C03642=1224.310,-102.269,-36.664,179.469,5.331,149.087
C03643=1224.305,-102.020,-36.674,179.472,5.331,149.087
C03644=1224.300,-101.770,-36.685,179.474,5.331,149.086
C03645=1224.294,-101.520,-36.695,179.476,5.332,149.085
C03646=1224.289,-101.271,-36.706,179.478,5.331,149.085
C03647=1224.283,-100.999,-36.717,179.481,5.332,149.084
C03648=1224.278,-100.728,-36.728,179.484,5.331,149.083
C03649=1224.272,-100.457,-36.740,179.486,5.331,149.082
C03650=1224.266,-100.186,-36.751,179.489,5.332,149.082
C03651=1224.261,-99.936,-36.761,179.491,5.331,149.081
C03652=1224.256,-99.687,-36.772,179.494,5.332,149.080
C03653=1224.251,-99.437,-36.783,179.496,5.332,149.079
C03654=1224.245,-99.187,-36.793,179.498,5.332,149.079
C03655=1224.240,-98.937,-36.804,179.500,5.332,149.078
C03656=1224.235,-98.688,-36.814,179.503,5.332,149.078
C03657=1224.230,-98.438,-36.825,179.505,5.332,149.077
C03658=1224.225,-98.189,-36.835,179.507,5.332,149.076
C03659=1224.220,-97.938,-36.846,179.510,5.332,149.075
C03660=1224.214,-97.689,-36.857,179.512,5.332,149.075
C03661=1224.209,-97.439,-36.868,179.514,5.332,149.074
C03662=1224.204,-97.190,-36.878,179.516,5.332,149.073
C03663=1224.199,-96.939,-36.888,179.519,5.332,149.073
C03664=1224.193,-96.690,-36.899,179.521,5.332,149.072
C03665=1224.188,-96.440,-36.910,179.523,5.333,149.071
C03666=1224.183,-96.191,-36.920,179.525,5.332,149.071
C03667=1224.178,-95.941,-36.931,179.528,5.333,149.070
C03668=1224.173,-95.691,-36.942,179.530,5.332,149.069
C03669=1224.168,-95.441,-36.952,179.533,5.333,149.069
C03670=1224.162,-95.192,-36.963,179.535,5.332,149.068
C03671=1224.157,-94.942,-36.974,179.538,5.333,149.067
C03672=1224.152,-94.692,-36.984,179.540,5.333,149.066
C03673=1224.147,-94.443,-36.995,179.542,5.333,149.066
C03674=1224.141,-94.193,-37.006,179.544,5.333,149.065
C03675=1224.136,-93.943,-37.016,179.547,5.333,149.064
C03676=1224.130,-93.694,-37.027,179.549,5.333,149.064
C03677=1224.125,-93.444,-37.038,179.551,5.334,149.063
C03678=1224.120,-93.195,-37.049,179.554,5.333,149.062
C03679=1224.115,-92.944,-37.059,179.556,5.334,149.062
C03680=1224.110,-92.694,-37.070,179.558,5.333,149.061
C03681=1224.105,-92.445,-37.081,179.561,5.334,149.060
C03682=1224.100,-92.195,-37.092,179.563,5.333,149.059
C03683=1224.094,-91.946,-37.102,179.566,5.334,149.059
C03684=1224.089,-91.696,-37.114,179.568,5.333,149.058
C03685=1224.083,-91.446,-37.124,179.571,5.334,149.057
C03686=1224.078,-91.196,-37.135,179.573,5.334,149.057
C03687=1224.073,-90.946,-37.146,179.575,5.334,149.056
C03688=1224.068,-90.697,-37.157,179.577,5.334,149.055
C03689=1224.063,-90.447,-37.167,179.580,5.334,149.055
C03690=1224.058,-90.198,-37.178,179.582,5.334,149.054
C03691=1224.053,-89.948,-37.189,179.584,5.334,149.053
C03692=1224.047,-89.698,-37.201,179.586,5.334,149.053
C03693=1224.042,-89.448,-37.211,179.589,5.335,149.052
C03694=1224.037,-89.199,-37.222,179.591,5.334,149.051
C03695=1224.032,-88.949,-37.232,179.594,5.335,149.050
C03696=1224.027,-88.699,-37.244,179.596,5.334,149.050
C03697=1224.022,-88.449,-37.254,179.599,5.335,149.049
C03698=1224.016,-88.200,-37.266,179.601,5.334,149.048
C03699=1224.011,-87.950,-37.276,179.603,5.335,149.048
C03700=1224.006,-87.701,-37.287,179.605,5.334,149.047
C03701=1224.001,-87.451,-37.298,179.608,5.335,149.046
C03702=1223.996,-87.201,-37.309,179.610,5.335,149.046
C03703=1223.990,-86.952,-37.321,179.612,5.335,149.045
C03704=1223.985,-86.701,-37.331,179.614,5.335,149.044
C03705=1223.980,-86.452,-37.342,179.617,5.335,149.044
C03706=1223.975,-86.202,-37.353,179.619,5.335,149.043
C03707=1223.969,-85.952,-37.365,179.622,5.336,149.042
C03708=1223.964,-85.703,-37.376,179.624,5.335,149.041
C03709=1223.959,-85.453,-37.386,179.627,5.336,149.041
C03710=1223.954,-85.204,-37.397,179.629,5.335,149.040
C03711=1223.949,-84.953,-37.408,179.631,5.336,149.039
C03712=1223.943,-84.704,-37.419,179.634,5.335,149.039
C03713=1223.938,-84.454,-37.431,179.636,5.336,149.038
C03714=1223.933,-84.204,-37.441,179.638,5.335,149.037
C03715=1223.927,-83.955,-37.453,179.641,5.336,149.036
C03716=1223.923,-83.705,-37.464,179.644,5.336,149.036
C03717=1223.918,-83.455,-37.475,179.645,5.336,149.035
C03718=1223.912,-83.206,-37.486,179.648,5.337,149.035
C03719=1223.907,-82.956,-37.497,179.650,5.337,149.034
C03720=1223.902,-82.706,-37.508,179.653,5.337,149.033
C03721=1223.897,-82.457,-37.519,179.655,5.337,149.032
C03722=1223.892,-82.207,-37.530,179.657,5.337,149.032
C03723=1223.886,-81.957,-37.541,179.660,5.337,149.031
C03724=1223.882,-81.707,-37.553,179.662,5.337,149.030
C03725=1223.876,-81.458,-37.564,179.664,5.337,149.030
C03726=1223.870,-81.208,-37.575,179.667,5.337,149.029
C03727=1223.866,-80.958,-37.586,179.669,5.337,149.028
C03728=1223.861,-80.709,-37.597,179.672,5.337,149.027
C03729=1223.855,-80.459,-37.609,179.674,5.337,149.027
C03730=1223.850,-80.209,-37.620,179.676,5.337,149.026
C03731=1223.845,-79.959,-37.631,179.679,5.337,149.025
C03732=1223.839,-79.710,-37.642,179.681,5.338,149.025
C03733=1223.835,-79.461,-37.654,179.683,5.337,149.024
C03734=1223.829,-79.211,-37.665,179.686,5.338,149.023
C03735=1223.824,-78.961,-37.676,179.688,5.338,149.023
C03736=1223.819,-78.711,-37.687,179.690,5.338,149.022
C03737=1223.814,-78.462,-37.699,179.692,5.338,149.021
C03738=1223.809,-78.212,-37.710,179.695,5.338,149.021
C03739=1223.804,-77.963,-37.721,179.697,5.338,149.020
C03740=1223.798,-77.712,-37.732,179.700,5.338,149.019
C03741=1223.793,-77.463,-37.744,179.702,5.339,149.018
C03742=1223.788,-77.213,-37.755,179.705,5.338,149.018
C03743=1223.783,-76.963,-37.767,179.707,5.339,149.017
C03744=1223.778,-76.714,-37.778,179.709,5.339,149.016
C03745=1223.772,-76.464,-37.790,179.712,5.339,149.016
C03746=1223.767,-76.214,-37.800,179.714,5.339,149.015
C03747=1223.762,-75.964,-37.812,179.717,5.339,149.014
C03748=1223.757,-75.715,-37.823,179.719,5.339,149.014
C03749=1223.751,-75.465,-37.835,179.722,5.339,149.013
C03750=1223.746,-75.216,-37.846,179.724,5.339,149.012
C03751=1223.741,-74.945,-37.858,179.726,5.339,149.011
C03752=1223.735,-74.675,-37.871,179.729,5.340,149.011
C03753=1223.729,-74.404,-37.883,179.731,5.339,149.010
C03754=1223.723,-74.134,-37.896,179.734,5.339,149.009
C03755=1223.719,-73.885,-37.907,179.736,5.339,149.009
C03756=1223.713,-73.635,-37.919,179.738,5.340,149.008
C03757=1223.708,-73.385,-37.930,179.741,5.340,149.007
C03758=1223.703,-73.135,-37.941,179.743,5.340,149.006
C03759=1223.698,-72.885,-37.953,179.746,5.341,149.006
C03760=1223.692,-72.636,-37.964,179.748,5.340,149.005
C03761=1223.687,-72.386,-37.976,179.751,5.341,149.004
C03762=1223.682,-72.136,-37.987,179.753,5.340,149.004
C03763=1223.677,-71.887,-37.999,179.755,5.341,149.003
C03764=1223.672,-71.637,-38.011,179.758,5.340,149.002
C03765=1223.667,-71.387,-38.022,179.760,5.341,149.001
C03766=1223.661,-71.138,-38.033,179.762,5.340,149.001
C03767=1223.656,-70.888,-38.045,179.765,5.341,149.000
C03768=1223.651,-70.638,-38.057,179.768,5.341,148.999
C03769=1223.646,-70.389,-38.068,179.770,5.341,148.999
C03770=1223.641,-70.139,-38.080,179.772,5.342,148.998
C03771=1223.635,-69.889,-38.092,179.774,5.341,148.997
C03772=1223.630,-69.640,-38.103,179.777,5.342,148.997
C03773=1223.625,-69.390,-38.114,179.779,5.341,148.996
C03774=1223.620,-69.141,-38.126,179.782,5.342,148.995
C03775=1223.615,-68.891,-38.138,179.784,5.341,148.994
C03776=1223.610,-68.641,-38.150,179.787,5.342,148.994
C03777=1223.605,-68.391,-38.162,179.789,5.342,148.993
C03778=1223.599,-68.142,-38.173,179.791,5.342,148.992
C03779=1223.595,-67.892,-38.185,179.794,5.342,148.992
C03780=1223.589,-67.642,-38.197,179.796,5.342,148.991
C03781=1223.584,-67.393,-38.207,179.799,5.343,148.990
C03782=1223.579,-67.143,-38.219,179.800,5.343,148.990
C03783=1223.573,-66.893,-38.231,179.803,5.343,148.989
C03784=1223.569,-66.644,-38.243,179.805,5.343,148.988
C03785=1223.563,-66.394,-38.255,179.808,5.343,148.988
C03786=1223.559,-66.145,-38.266,179.810,5.343,148.987
C03787=1223.553,-65.895,-38.278,179.813,5.343,148.986
C03788=1223.548,-65.645,-38.290,179.815,5.343,148.985
C03789=1223.543,-65.395,-38.302,179.817,5.343,148.985
C03790=1223.538,-65.145,-38.313,179.820,5.344,148.984
C03791=1223.532,-64.896,-38.326,179.822,5.344,148.983
C03792=1223.527,-64.647,-38.337,179.825,5.344,148.983
C03793=1223.522,-64.397,-38.349,179.827,5.344,148.982
C03794=1223.516,-64.147,-38.361,179.830,5.344,148.981
C03795=1223.512,-63.897,-38.372,179.832,5.344,148.981
C03796=1223.507,-63.648,-38.385,179.834,5.344,148.980
C03797=1223.501,-63.398,-38.396,179.837,5.345,148.979
C03798=1223.496,-63.149,-38.408,179.839,5.344,148.978
C03799=1223.491,-62.899,-38.420,179.842,5.345,148.978
C03800=1223.486,-62.649,-38.432,179.844,5.344,148.977
C03801=1223.480,-62.399,-38.444,179.846,5.345,148.976
C03802=1223.476,-62.150,-38.455,179.849,5.345,148.976
C03803=1223.470,-61.900,-38.467,179.851,5.345,148.975
C03804=1223.465,-61.650,-38.480,179.853,5.345,148.974
C03805=1223.460,-61.401,-38.491,179.856,5.345,148.973
C03806=1223.455,-61.151,-38.503,179.859,5.346,148.973
C03807=1223.450,-60.902,-38.516,179.861,5.345,148.972
C03808=1223.445,-60.652,-38.528,179.863,5.346,148.971
C03809=1223.440,-60.402,-38.539,179.865,5.345,148.971
C03810=1223.434,-60.152,-38.551,179.868,5.346,148.970
C03811=1223.429,-59.903,-38.563,179.870,5.346,148.969
C03812=1223.424,-59.653,-38.575,179.873,5.346,148.969
C03813=1223.419,-59.403,-38.587,179.876,5.347,148.968
C03814=1223.414,-59.154,-38.599,179.878,5.346,148.967
C03815=1223.409,-58.904,-38.611,179.880,5.347,148.966
C03816=1223.403,-58.655,-38.624,179.882,5.346,148.966
C03817=1223.399,-58.405,-38.635,179.885,5.347,148.965
C03818=1223.393,-58.155,-38.647,179.887,5.346,148.964
C03819=1223.388,-57.906,-38.659,179.890,5.347,148.964
C03820=1223.383,-57.656,-38.671,179.893,5.347,148.963
C03821=1223.377,-57.406,-38.683,179.895,5.347,148.962
C03822=1223.373,-57.157,-38.695,179.897,5.348,148.962
C03823=1223.368,-56.907,-38.707,179.899,5.348,148.961
C03824=1223.362,-56.658,-38.720,179.902,5.348,148.960
C03825=1223.357,-56.408,-38.732,179.904,5.348,148.960
C03826=1223.352,-56.158,-38.744,179.906,5.348,148.959
C03827=1223.346,-55.908,-38.756,179.909,5.349,148.958
C03828=1223.342,-55.659,-38.767,179.911,5.348,148.957
C03829=1223.337,-55.409,-38.780,179.914,5.349,148.957
C03830=1223.332,-55.159,-38.792,179.916,5.348,148.956
C03831=1223.327,-54.910,-38.805,179.918,5.349,148.955
C03832=1223.321,-54.660,-38.817,179.921,5.349,148.955
C03833=1223.316,-54.410,-38.829,179.923,5.349,148.954
C03834=1223.311,-54.161,-38.841,179.926,5.350,148.953
C03835=1223.306,-53.911,-38.853,179.928,5.349,148.953
C03836=1223.301,-53.661,-38.865,179.931,5.350,148.952
C03837=1223.296,-53.412,-38.878,179.933,5.349,148.951
C03838=1223.290,-53.162,-38.889,179.935,5.350,148.950
C03839=1223.285,-52.913,-38.902,179.938,5.350,148.950
C03840=1223.280,-52.662,-38.914,179.940,5.350,148.949
C03841=1223.275,-52.413,-38.927,179.943,5.350,148.948
C03842=1223.270,-52.163,-38.939,179.945,5.350,148.948
C03843=1223.265,-51.914,-38.951,179.948,5.351,148.947
C03844=1223.260,-51.665,-38.963,179.950,5.351,148.946
C03845=1223.255,-51.415,-38.975,179.952,5.351,148.946
C03846=1223.250,-51.165,-38.988,179.955,5.351,148.945
C03847=1223.244,-50.915,-39.000,179.957,5.351,148.944
C03848=1223.239,-50.666,-39.012,179.960,5.351,148.943
C03849=1223.234,-50.415,-39.025,179.962,5.352,148.943
C03850=1223.229,-50.166,-39.037,179.964,5.351,148.942
C03851=1223.224,-49.917,-39.050,179.967,5.352,148.941
C03852=1223.219,-49.667,-39.062,179.969,5.352,148.941
C03853=1223.214,-49.418,-39.074,179.972,5.352,148.940
C03854=1223.208,-49.168,-39.087,179.975,5.353,148.939
C03855=1223.203,-48.898,-39.100,179.977,5.352,148.938
C03856=1223.197,-48.628,-39.114,179.979,5.353,148.938
C03857=1223.191,-48.358,-39.127,179.982,5.353,148.937
C03858=1223.186,-48.088,-39.140,179.985,5.352,148.936
C03859=1223.181,-47.839,-39.153,179.987,5.353,148.935
C03860=1223.176,-47.589,-39.165,179.990,5.353,148.935
C03861=1223.171,-47.340,-39.178,179.992,5.353,148.934
C03862=1223.166,-47.090,-39.191,179.995,5.354,148.933
C03863=1223.161,-46.840,-39.202,179.997,5.353,148.933
C03864=1223.156,-46.591,-39.215,179.999,5.354,148.932
C03865=1223.151,-46.341,-39.228,-179.998,5.354,148.931
C03866=1223.145,-46.091,-39.239,-179.996,5.354,148.931
C03867=1223.140,-45.842,-39.252,-179.993,5.354,148.930
C03868=1223.136,-45.592,-39.265,-179.991,5.354,148.929
C03869=1223.130,-45.343,-39.278,-179.988,5.354,148.928
C03870=1223.124,-45.092,-39.290,-179.986,5.355,148.928
C03871=1223.119,-44.843,-39.303,-179.984,5.355,148.927
C03872=1223.114,-44.594,-39.315,-179.981,5.355,148.926
C03873=1223.109,-44.344,-39.328,-179.978,5.356,148.926
C03874=1223.104,-44.094,-39.340,-179.976,5.355,148.925
C03875=1223.099,-43.845,-39.353,-179.974,5.356,148.924
C03876=1223.094,-43.595,-39.365,-179.972,5.355,148.924
C03877=1223.089,-43.345,-39.378,-179.969,5.356,148.923
C03878=1223.084,-43.096,-39.391,-179.966,5.356,148.922
C03879=1223.079,-42.846,-39.403,-179.964,5.356,148.921
C03880=1223.074,-42.597,-39.415,-179.961,5.357,148.921
C03881=1223.068,-42.346,-39.429,-179.959,5.356,148.920
C03882=1223.063,-42.097,-39.442,-179.957,5.357,148.919
C03883=1223.058,-41.848,-39.454,-179.954,5.357,148.919
C03884=1223.053,-41.598,-39.467,-179.952,5.357,148.918
C03885=1223.048,-41.348,-39.480,-179.949,5.357,148.917
C03886=1223.043,-41.098,-39.492,-179.947,5.358,148.916
C03887=1223.038,-40.849,-39.504,-179.945,5.358,148.916
C03888=1223.032,-40.599,-39.517,-179.942,5.358,148.915
C03889=1223.027,-40.349,-39.530,-179.940,5.358,148.914
C03890=1223.022,-40.100,-39.543,-179.937,5.358,148.914
C03891=1223.017,-39.851,-39.556,-179.934,5.359,148.913
C03892=1223.012,-39.602,-39.568,-179.932,5.358,148.912
C03893=1223.008,-39.351,-39.581,-179.930,5.359,148.912
C03894=1223.002,-39.102,-39.594,-179.927,5.359,148.911
C03895=1222.997,-38.853,-39.607,-179.925,5.359,148.910
C03896=1222.992,-38.602,-39.619,-179.923,5.360,148.910
C03897=1222.987,-38.353,-39.632,-179.921,5.359,148.909
C03898=1222.982,-38.103,-39.644,-179.918,5.360,148.908
C03899=1222.976,-37.854,-39.658,-179.915,5.360,148.908
C03900=1222.971,-37.604,-39.671,-179.913,5.360,148.907
C03901=1222.966,-37.354,-39.683,-179.911,5.361,148.906
C03902=1222.961,-37.105,-39.696,-179.908,5.361,148.906
C03903=1222.956,-36.855,-39.709,-179.906,5.361,148.905
C03904=1222.951,-36.605,-39.722,-179.903,5.361,148.904
C03905=1222.945,-36.356,-39.735,-179.901,5.361,148.903
C03906=1222.941,-36.106,-39.748,-179.899,5.361,148.903
C03907=1222.935,-35.856,-39.761,-179.896,5.362,148.902
C03908=1222.930,-35.607,-39.773,-179.894,5.362,148.901
C03909=1222.925,-35.357,-39.786,-179.891,5.362,148.901
C03910=1222.920,-35.108,-39.799,-179.888,5.363,148.900
C03911=1222.914,-34.858,-39.812,-179.886,5.362,148.899
C03912=1222.910,-34.609,-39.826,-179.884,5.363,148.899
C03913=1222.905,-34.359,-39.838,-179.881,5.363,148.898
C03914=1222.899,-34.110,-39.852,-179.879,5.363,148.897
C03915=1222.895,-33.860,-39.865,-179.876,5.363,148.896
C03916=1222.890,-33.610,-39.877,-179.874,5.364,148.896
C03917=1222.884,-33.361,-39.890,-179.872,5.364,148.895
C03918=1222.879,-33.111,-39.903,-179.869,5.364,148.894
C03919=1222.874,-32.861,-39.916,-179.867,5.364,148.894
C03920=1222.870,-32.611,-39.929,-179.864,5.364,148.893
C03921=1222.864,-32.362,-39.942,-179.861,5.365,148.892
C03922=1222.859,-32.113,-39.955,-179.859,5.364,148.892
C03923=1222.854,-31.863,-39.968,-179.857,5.365,148.891
C03924=1222.848,-31.613,-39.982,-179.854,5.365,148.890
C03925=1222.843,-31.364,-39.994,-179.852,5.365,148.889
C03926=1222.838,-31.114,-40.008,-179.849,5.366,148.889
C03927=1222.833,-30.864,-40.020,-179.847,5.366,148.888
C03928=1222.829,-30.615,-40.034,-179.845,5.366,148.887
C03929=1222.823,-30.365,-40.047,-179.842,5.366,148.887
C03930=1222.818,-30.116,-40.060,-179.839,5.367,148.886
C03931=1222.813,-29.866,-40.073,-179.837,5.366,148.885
C03932=1222.807,-29.617,-40.086,-179.835,5.367,148.885
C03933=1222.803,-29.367,-40.100,-179.832,5.367,148.884
C03934=1222.797,-29.117,-40.113,-179.830,5.367,148.883
C03935=1222.793,-28.867,-40.126,-179.827,5.368,148.882
C03936=1222.788,-28.618,-40.138,-179.824,5.368,148.882
C03937=1222.782,-28.369,-40.152,-179.822,5.368,148.881
C03938=1222.778,-28.119,-40.165,-179.820,5.368,148.880
C03939=1222.772,-27.869,-40.178,-179.817,5.369,148.880
C03940=1222.767,-27.619,-40.191,-179.815,5.368,148.879
C03941=1222.762,-27.370,-40.205,-179.812,5.369,148.878
C03942=1222.757,-27.120,-40.218,-179.810,5.369,148.878
C03943=1222.752,-26.871,-40.231,-179.808,5.369,148.877
C03944=1222.747,-26.621,-40.244,-179.805,5.370,148.876
C03945=1222.742,-26.372,-40.258,-179.802,5.370,148.875
C03946=1222.737,-26.122,-40.271,-179.800,5.370,148.875
C03947=1222.731,-25.872,-40.284,-179.798,5.370,148.874
C03948=1222.727,-25.623,-40.298,-179.795,5.371,148.873
C03949=1222.721,-25.373,-40.311,-179.793,5.370,148.873
C03950=1222.716,-25.124,-40.324,-179.790,5.371,148.872
C03951=1222.711,-24.874,-40.338,-179.787,5.371,148.871
C03952=1222.705,-24.625,-40.351,-179.785,5.371,148.871
C03953=1222.701,-24.375,-40.364,-179.783,5.372,148.870
C03954=1222.695,-24.126,-40.378,-179.780,5.372,148.869
C03955=1222.691,-23.876,-40.391,-179.778,5.372,148.869
C03956=1222.685,-23.627,-40.405,-179.775,5.372,148.868
C03957=1222.681,-23.377,-40.418,-179.773,5.373,148.867
C03958=1222.675,-23.127,-40.431,-179.771,5.372,148.866
C03959=1222.670,-22.858,-40.445,-179.768,5.373,148.866
C03960=1222.665,-22.589,-40.460,-179.765,5.373,148.865
C03961=1222.659,-22.318,-40.474,-179.762,5.374,148.864
C03962=1222.653,-22.050,-40.489,-179.759,5.374,148.863
C03963=1222.649,-21.800,-40.502,-179.757,5.374,148.863
C03964=1222.643,-21.551,-40.516,-179.755,5.374,148.862
C03965=1222.638,-21.301,-40.529,-179.752,5.375,148.861
C03966=1222.633,-21.051,-40.543,-179.750,5.374,148.861
C03967=1222.628,-20.802,-40.556,-179.747,5.375,148.860
C03968=1222.623,-20.552,-40.570,-179.745,5.375,148.859
C03969=1222.618,-20.302,-40.583,-179.743,5.375,148.859
C03970=1222.613,-20.053,-40.597,-179.740,5.376,148.858
C03971=1222.607,-19.803,-40.610,-179.737,5.376,148.857
C03972=1222.603,-19.554,-40.624,-179.735,5.376,148.856
C03973=1222.597,-19.304,-40.637,-179.732,5.376,148.856
C03974=1222.592,-19.055,-40.651,-179.730,5.377,148.855
C03975=1222.588,-18.805,-40.664,-179.728,5.377,148.854
C03976=1222.582,-18.556,-40.678,-179.725,5.377,148.854
C03977=1222.578,-18.306,-40.691,-179.722,5.378,148.853
C03978=1222.572,-18.057,-40.705,-179.720,5.378,148.852
C03979=1222.567,-17.807,-40.719,-179.718,5.378,148.852
C03980=1222.562,-17.558,-40.732,-179.715,5.378,148.851
C03981=1222.557,-17.308,-40.746,-179.713,5.379,148.850
C03982=1222.552,-17.057,-40.760,-179.711,5.379,148.850
C03983=1222.547,-16.809,-40.773,-179.708,5.379,148.849
C03984=1222.542,-16.558,-40.787,-179.705,5.380,148.848
C03985=1222.536,-16.309,-40.801,-179.703,5.380,148.848
C03986=1222.532,-16.060,-40.814,-179.701,5.380,148.847
C03987=1222.527,-15.810,-40.828,-179.698,5.381,148.846
C03988=1222.521,-15.561,-40.842,-179.696,5.380,148.846
C03989=1222.516,-15.311,-40.856,-179.693,5.381,148.845
C03990=1222.511,-15.062,-40.869,-179.691,5.381,148.844
C03991=1222.506,-14.812,-40.883,-179.688,5.382,148.844
C03992=1222.501,-14.562,-40.897,-179.686,5.381,148.843
C03993=1222.496,-14.313,-40.910,-179.683,5.382,148.842
C03994=1222.491,-14.063,-40.924,-179.681,5.382,148.841
C03995=1222.486,-13.814,-40.938,-179.679,5.382,148.841
C03996=1222.480,-13.564,-40.952,-179.676,5.383,148.840
C03997=1222.476,-13.314,-40.965,-179.673,5.383,148.839
C03998=1222.471,-13.065,-40.980,-179.671,5.384,148.839
C03999=1222.465,-12.815,-40.993,-179.669,5.383,148.838
C04000=1222.460,-12.565,-41.007,-179.666,5.384,148.837
C04001=1222.456,-12.316,-41.021,-179.663,5.384,148.837
C04002=1222.451,-12.067,-41.035,-179.661,5.384,148.836
C04003=1222.445,-11.817,-41.048,-179.658,5.385,148.835
C04004=1222.440,-11.567,-41.062,-179.656,5.385,148.835
C04005=1222.436,-11.318,-41.076,-179.653,5.386,148.834
C04006=1222.431,-11.069,-41.090,-179.651,5.385,148.833
C04007=1222.425,-10.818,-41.104,-179.648,5.386,148.832
C04008=1222.420,-10.569,-41.117,-179.646,5.386,148.832
C04009=1222.415,-10.320,-41.132,-179.644,5.386,148.831
C04010=1222.411,-10.070,-41.145,-179.641,5.387,148.830
C04011=1222.405,-9.821,-41.159,-179.638,5.387,148.830
C04012=1222.400,-9.571,-41.173,-179.636,5.388,148.829
C04013=1222.395,-9.321,-41.187,-179.634,5.387,148.828
C04014=1222.390,-9.071,-41.201,-179.631,5.388,148.828
C04015=1222.385,-8.823,-41.215,-179.628,5.388,148.827
C04016=1222.380,-8.573,-41.229,-179.626,5.389,148.826
C04017=1222.375,-8.323,-41.243,-179.624,5.388,148.826
C04018=1222.370,-8.074,-41.257,-179.621,5.389,148.825
C04019=1222.364,-7.824,-41.271,-179.618,5.389,148.824
C04020=1222.359,-7.574,-41.285,-179.616,5.389,148.823
C04021=1222.355,-7.324,-41.299,-179.614,5.390,148.823
C04022=1222.350,-7.076,-41.313,-179.611,5.390,148.822
C04023=1222.345,-6.826,-41.327,-179.608,5.391,148.821
C04024=1222.340,-6.576,-41.341,-179.606,5.390,148.821
C04025=1222.335,-6.327,-41.356,-179.604,5.391,148.820
C04026=1222.329,-6.078,-41.369,-179.601,5.391,148.819
C04027=1222.324,-5.828,-41.384,-179.598,5.392,148.819
C04028=1222.319,-5.578,-41.398,-179.597,5.392,148.818
C04029=1222.314,-5.329,-41.412,-179.594,5.393,148.817
C04030=1222.309,-5.079,-41.425,-179.591,5.393,148.817
C04031=1222.304,-4.829,-41.440,-179.589,5.394,148.816
C04032=1222.299,-4.580,-41.453,-179.587,5.393,148.815
C04033=1222.294,-4.330,-41.468,-179.584,5.394,148.815
C04034=1222.289,-4.080,-41.482,-179.581,5.394,148.814
C04035=1222.284,-3.831,-41.496,-179.579,5.395,148.813
C04036=1222.279,-3.582,-41.510,-179.577,5.395,148.813
C04037=1222.274,-3.332,-41.524,-179.574,5.395,148.812
C04038=1222.269,-3.082,-41.539,-179.571,5.396,148.811
C04039=1222.264,-2.832,-41.553,-179.569,5.396,148.811
C04040=1222.259,-2.583,-41.567,-179.567,5.396,148.810
C04041=1222.254,-2.334,-41.581,-179.564,5.396,148.809
C04042=1222.249,-2.085,-41.596,-179.561,5.397,148.808
C04043=1222.244,-1.835,-41.610,-179.559,5.397,148.808
C04044=1222.239,-1.585,-41.625,-179.556,5.397,148.807
C04045=1222.233,-1.336,-41.639,-179.554,5.398,148.806
C04046=1222.229,-1.087,-41.653,-179.551,5.398,148.806
C04047=1222.224,-0.837,-41.667,-179.548,5.399,148.805
C04048=1222.219,-0.587,-41.681,-179.546,5.398,148.804
C04049=1222.214,-0.337,-41.696,-179.544,5.399,148.804
C04050=1222.209,-0.088,-41.710,-179.541,5.399,148.803
C04051=1222.203,0.161,-41.724,-179.538,5.400,148.802
C04052=1222.198,0.411,-41.738,-179.536,5.400,148.802
C04053=1222.194,0.660,-41.753,-179.534,5.400,148.801
C04054=1222.189,0.910,-41.767,-179.531,5.401,148.800
C04055=1222.184,1.160,-41.782,-179.528,5.401,148.800
C04056=1222.179,1.409,-41.796,-179.526,5.401,148.799
C04057=1222.173,1.659,-41.811,-179.524,5.401,148.798
C04058=1222.167,1.908,-41.825,-179.522,5.402,148.798
C04059=1222.163,2.157,-41.840,-179.519,5.403,148.797
C04060=1222.158,2.407,-41.854,-179.517,5.402,148.796
C04061=1222.153,2.657,-41.868,-179.514,5.403,148.796
C04062=1222.148,2.906,-41.883,-179.512,5.403,148.795
C04063=1222.143,3.175,-41.898,-179.508,5.404,148.794
C04064=1222.138,3.444,-41.914,-179.506,5.404,148.793
C04065=1222.131,3.714,-41.930,-179.503,5.405,148.793
C04066=1222.126,3.982,-41.945,-179.500,5.405,148.792
C04067=1222.121,4.232,-41.959,-179.498,5.405,148.791
C04068=1222.116,4.481,-41.974,-179.496,5.405,148.791
C04069=1222.111,4.730,-41.989,-179.493,5.406,148.790
C04070=1222.106,4.980,-42.003,-179.490,5.406,148.789
C04071=1222.101,5.230,-42.017,-179.488,5.407,148.789
C04072=1222.096,5.479,-42.033,-179.486,5.407,148.788
C04073=1222.091,5.729,-42.047,-179.483,5.407,148.787
C04074=1222.086,5.979,-42.061,-179.480,5.408,148.786
C04075=1222.081,6.228,-42.076,-179.478,5.408,148.786
C04076=1222.076,6.477,-42.090,-179.476,5.408,148.785
C04077=1222.071,6.727,-42.105,-179.473,5.408,148.784
C04078=1222.066,6.977,-42.120,-179.470,5.409,148.784
C04079=1222.060,7.226,-42.134,-179.468,5.410,148.783
C04080=1222.056,7.475,-42.149,-179.466,5.410,148.783
C04081=1222.051,7.724,-42.164,-179.463,5.410,148.782
C04082=1222.046,7.974,-42.178,-179.461,5.411,148.781
C04083=1222.040,8.224,-42.193,-179.458,5.411,148.780
C04084=1222.036,8.473,-42.208,-179.455,5.412,148.780
C04085=1222.031,8.723,-42.222,-179.453,5.412,148.779
C04086=1222.026,8.973,-42.236,-179.451,5.412,148.778
C04087=1222.020,9.222,-42.252,-179.448,5.412,148.778
C04088=1222.015,9.472,-42.266,-179.445,5.413,148.777
C04089=1222.011,9.721,-42.281,-179.443,5.414,148.776
C04090=1222.006,9.971,-42.295,-179.440,5.414,148.776
C04091=1222.000,10.220,-42.311,-179.438,5.414,148.775
C04092=1221.995,10.470,-42.325,-179.435,5.414,148.774
C04093=1221.990,10.719,-42.340,-179.433,5.415,148.774
C04094=1221.986,10.968,-42.355,-179.430,5.415,148.773
C04095=1221.980,11.218,-42.369,-179.427,5.416,148.772
C04096=1221.975,11.468,-42.384,-179.425,5.416,148.772
C04097=1221.970,11.717,-42.399,-179.423,5.416,148.771
C04098=1221.966,11.966,-42.414,-179.420,5.417,148.770
C04099=1221.960,12.216,-42.429,-179.418,5.418,148.770
C04100=1221.955,12.465,-42.444,-179.415,5.418,148.769
C04101=1221.951,12.715,-42.458,-179.413,5.418,148.768
C04102=1221.945,12.965,-42.473,-179.411,5.418,148.768
C04103=1221.940,13.214,-42.488,-179.408,5.419,148.767
C04104=1221.936,13.463,-42.503,-179.405,5.419,148.766
C04105=1221.930,13.713,-42.518,-179.403,5.420,148.766
C04106=1221.925,13.962,-42.533,-179.401,5.420,148.765
C04107=1221.921,14.212,-42.548,-179.398,5.420,148.764
C04108=1221.915,14.462,-42.562,-179.395,5.421,148.764
C04109=1221.911,14.711,-42.578,-179.393,5.421,148.763
C04110=1221.905,14.961,-42.593,-179.390,5.422,148.762
C04111=1221.900,15.211,-42.608,-179.388,5.421,148.762
C04112=1221.896,15.460,-42.622,-179.385,5.422,148.761
C04113=1221.890,15.710,-42.637,-179.383,5.423,148.760
C04114=1221.885,15.959,-42.652,-179.380,5.423,148.759
C04115=1221.881,16.208,-42.667,-179.377,5.424,148.759
C04116=1221.875,16.458,-42.682,-179.375,5.424,148.758
C04117=1221.870,16.707,-42.697,-179.373,5.424,148.758
C04118=1221.865,16.957,-42.712,-179.370,5.425,148.757
C04119=1221.860,17.206,-42.727,-179.368,5.425,148.756
C04120=1221.856,17.455,-42.742,-179.365,5.426,148.756
C04121=1221.850,17.705,-42.757,-179.362,5.426,148.755
C04122=1221.846,17.955,-42.772,-179.360,5.427,148.754
C04123=1221.840,18.204,-42.788,-179.358,5.427,148.754
C04124=1221.835,18.454,-42.802,-179.355,5.427,148.753
C04125=1221.830,18.703,-42.818,-179.352,5.428,148.752
C04126=1221.825,18.953,-42.833,-179.350,5.428,148.752
C04127=1221.820,19.203,-42.848,-179.347,5.429,148.751
C04128=1221.815,19.452,-42.863,-179.345,5.429,148.750
C04129=1221.810,19.701,-42.878,-179.342,5.429,148.749
C04130=1221.806,19.951,-42.894,-179.340,5.430,148.749
C04131=1221.801,20.201,-42.908,-179.338,5.430,148.748
C04132=1221.795,20.450,-42.924,-179.335,5.431,148.748
C04133=1221.791,20.699,-42.939,-179.332,5.431,148.747
C04134=1221.785,20.948,-42.954,-179.330,5.432,148.746
C04135=1221.780,21.198,-42.968,-179.328,5.432,148.746
C04136=1221.775,21.448,-42.984,-179.325,5.432,148.745
C04137=1221.771,21.697,-42.999,-179.322,5.433,148.744
C04138=1221.765,21.947,-43.015,-179.320,5.433,148.744
C04139=1221.760,22.196,-43.031,-179.317,5.434,148.743
C04140=1221.755,22.445,-43.045,-179.314,5.434,148.742
C04141=1221.750,22.695,-43.060,-179.312,5.435,148.742
C04142=1221.745,22.944,-43.075,-179.310,5.435,148.741
C04143=1221.740,23.194,-43.091,-179.308,5.436,148.740
C04144=1221.736,23.444,-43.106,-179.305,5.436,148.740
C04145=1221.730,23.693,-43.122,-179.302,5.437,148.739
C04146=1221.726,23.942,-43.137,-179.300,5.437,148.738
C04147=1221.720,24.191,-43.152,-179.297,5.438,148.738
C04148=1221.715,24.442,-43.168,-179.294,5.438,148.737
C04149=1221.710,24.691,-43.183,-179.292,5.438,148.736
C04150=1221.705,24.941,-43.198,-179.290,5.439,148.736
C04151=1221.700,25.190,-43.213,-179.287,5.439,148.735
C04152=1221.695,25.439,-43.229,-179.284,5.440,148.734
C04153=1221.691,25.689,-43.244,-179.282,5.440,148.734
C04154=1221.686,25.938,-43.260,-179.279,5.441,148.733
C04155=1221.680,26.188,-43.275,-179.277,5.442,148.732
C04156=1221.676,26.437,-43.290,-179.275,5.441,148.732
C04157=1221.671,26.687,-43.306,-179.272,5.442,148.731
C04158=1221.665,26.936,-43.322,-179.269,5.442,148.730
C04159=1221.661,27.185,-43.337,-179.267,5.443,148.730
C04160=1221.655,27.435,-43.353,-179.264,5.443,148.729
C04161=1221.651,27.685,-43.368,-179.262,5.444,148.728
C04162=1221.646,27.934,-43.383,-179.259,5.445,148.728
C04163=1221.641,28.183,-43.399,-179.257,5.444,148.727
C04164=1221.635,28.433,-43.415,-179.254,5.445,148.726
C04165=1221.631,28.683,-43.430,-179.252,5.445,148.726
C04166=1221.626,28.932,-43.446,-179.249,5.446,148.725
C04167=1221.620,29.201,-43.463,-179.246,5.446,148.724
C04168=1221.615,29.469,-43.478,-179.244,5.447,148.724
C04169=1221.609,29.738,-43.495,-179.241,5.448,148.723
C04170=1221.604,30.006,-43.512,-179.238,5.448,148.722
C04171=1221.599,30.256,-43.528,-179.236,5.449,148.722
C04172=1221.594,30.505,-43.543,-179.233,5.449,148.721
C04173=1221.589,30.755,-43.559,-179.230,5.450,148.720
C04174=1221.584,31.005,-43.575,-179.228,5.450,148.720
C04175=1221.579,31.254,-43.590,-179.226,5.451,148.719
C04176=1221.574,31.503,-43.605,-179.223,5.452,148.718
C04177=1221.569,31.752,-43.622,-179.221,5.451,148.718
C04178=1221.564,32.002,-43.638,-179.218,5.452,148.717
C04179=1221.559,32.252,-43.653,-179.216,5.452,148.716
C04180=1221.554,32.501,-43.668,-179.213,5.453,148.716
C04181=1221.550,32.751,-43.684,-179.210,5.454,148.715
C04182=1221.544,33.000,-43.700,-179.208,5.454,148.714
C04183=1221.539,33.249,-43.716,-179.205,5.455,148.714
C04184=1221.535,33.499,-43.731,-179.202,5.455,148.713
C04185=1221.530,33.748,-43.747,-179.200,5.456,148.713
C04186=1221.524,33.998,-43.763,-179.198,5.456,148.712
C04187=1221.520,34.248,-43.779,-179.196,5.456,148.711
C04188=1221.514,34.497,-43.795,-179.193,5.457,148.711
C04189=1221.510,34.746,-43.810,-179.190,5.458,148.710
C04190=1221.505,34.996,-43.826,-179.188,5.458,148.709
C04191=1221.500,35.245,-43.841,-179.185,5.459,148.709
C04192=1221.495,35.495,-43.857,-179.182,5.459,148.708
C04193=1221.490,35.744,-43.874,-179.180,5.460,148.707
C04194=1221.484,35.994,-43.889,-179.178,5.461,148.707
C04195=1221.480,36.243,-43.905,-179.175,5.461,148.706
C04196=1221.475,36.492,-43.921,-179.172,5.462,148.705
C04197=1221.470,36.741,-43.937,-179.170,5.461,148.705
C04198=1221.465,36.992,-43.952,-179.168,5.462,148.704
C04199=1221.460,37.241,-43.968,-179.165,5.463,148.703
C04200=1221.455,37.490,-43.985,-179.162,5.463,148.703
C04201=1221.450,37.740,-44.000,-179.160,5.464,148.702
C04202=1221.444,37.989,-44.016,-179.157,5.465,148.702
C04203=1221.441,38.238,-44.032,-179.155,5.465,148.701
C04204=1221.435,38.488,-44.048,-179.152,5.466,148.700
C04205=1221.431,38.738,-44.064,-179.150,5.466,148.700
C04206=1221.425,38.987,-44.080,-179.147,5.467,148.699
C04207=1221.420,39.236,-44.095,-179.144,5.467,148.698
C04208=1221.416,39.486,-44.112,-179.142,5.468,148.698
C04209=1221.410,39.735,-44.128,-179.140,5.468,148.697
C04210=1221.405,39.985,-44.144,-179.137,5.468,148.696
C04211=1221.400,40.234,-44.160,-179.135,5.469,148.696
C04212=1221.396,40.484,-44.176,-179.132,5.470,148.695
C04213=1221.390,40.733,-44.192,-179.129,5.470,148.694
C04214=1221.385,40.982,-44.208,-179.127,5.471,148.694
C04215=1221.380,41.232,-44.224,-179.124,5.471,148.693
C04216=1221.375,41.481,-44.240,-179.122,5.472,148.692
C04217=1221.370,41.731,-44.256,-179.119,5.472,148.692
C04218=1221.365,41.980,-44.272,-179.117,5.473,148.691
C04219=1221.361,42.230,-44.288,-179.114,5.474,148.691
C04220=1221.355,42.479,-44.305,-179.111,5.474,148.690
C04221=1221.351,42.729,-44.321,-179.109,5.475,148.689
C04222=1221.346,42.978,-44.337,-179.106,5.475,148.689
C04223=1221.341,43.228,-44.353,-179.104,5.475,148.688
C04224=1221.336,43.477,-44.369,-179.102,5.476,148.687
C04225=1221.331,43.727,-44.385,-179.099,5.477,148.687
C04226=1221.326,43.976,-44.401,-179.097,5.477,148.686
C04227=1221.321,44.226,-44.417,-179.094,5.478,148.685
C04228=1221.316,44.474,-44.434,-179.091,5.478,148.685
C04229=1221.312,44.724,-44.450,-179.089,5.479,148.684
C04230=1221.306,44.973,-44.466,-179.086,5.479,148.683
C04231=1221.302,45.223,-44.483,-179.084,5.480,148.683
C04232=1221.296,45.472,-44.498,-179.081,5.481,148.682
C04233=1221.292,45.722,-44.515,-179.079,5.481,148.682
C04234=1221.286,45.971,-44.530,-179.076,5.482,148.681
C04235=1221.282,46.221,-44.547,-179.073,5.483,148.680
C04236=1221.277,46.469,-44.563,-179.071,5.483,148.680
C04237=1221.272,46.719,-44.579,-179.068,5.484,148.679
C04238=1221.266,46.969,-44.596,-179.066,5.484,148.678
C04239=1221.262,47.218,-44.613,-179.063,5.485,148.678
C04240=1221.256,47.467,-44.628,-179.061,5.486,148.677
C04241=1221.252,47.717,-44.645,-179.058,5.486,148.676
C04242=1221.247,47.966,-44.661,-179.055,5.487,148.676
C04243=1221.242,48.216,-44.677,-179.053,5.487,148.675
C04244=1221.238,48.465,-44.694,-179.050,5.488,148.674
C04245=1221.232,48.714,-44.710,-179.048,5.488,148.674
C04246=1221.227,48.964,-44.727,-179.046,5.489,148.673
C04247=1221.222,49.213,-44.743,-179.043,5.489,148.673
C04248=1221.217,49.463,-44.760,-179.041,5.490,148.672
C04249=1221.212,49.712,-44.775,-179.038,5.490,148.671
C04250=1221.207,49.962,-44.792,-179.035,5.491,148.671
C04251=1221.203,50.211,-44.809,-179.033,5.491,148.670
C04252=1221.197,50.460,-44.826,-179.031,5.492,148.670
C04253=1221.192,50.710,-44.842,-179.028,5.493,148.669
C04254=1221.187,50.959,-44.858,-179.025,5.493,148.668
C04255=1221.183,51.209,-44.875,-179.023,5.494,148.668
C04256=1221.178,51.458,-44.891,-179.020,5.495,148.667
C04257=1221.173,51.707,-44.908,-179.017,5.495,148.666
C04258=1221.168,51.957,-44.924,-179.015,5.496,148.666
C04259=1221.163,52.207,-44.941,-179.013,5.497,148.665
C04260=1221.158,52.456,-44.957,-179.010,5.497,148.664
C04261=1221.154,52.705,-44.974,-179.007,5.498,148.664
C04262=1221.148,52.954,-44.991,-179.005,5.498,148.663
C04263=1221.143,53.204,-45.007,-179.002,5.499,148.662
C04264=1221.139,53.454,-45.023,-179.000,5.500,148.662
C04265=1221.134,53.702,-45.040,-178.997,5.500,148.661
C04266=1221.128,53.952,-45.057,-178.995,5.501,148.661
C04267=1221.124,54.202,-45.074,-178.992,5.502,148.660
C04268=1221.119,54.451,-45.090,-178.989,5.502,148.659
C04269=1221.114,54.700,-45.106,-178.987,5.503,148.659
C04270=1221.109,54.950,-45.124,-178.985,5.504,148.658
C04271=1221.104,55.218,-45.141,-178.982,5.504,148.657
C04272=1221.099,55.487,-45.159,-178.979,5.504,148.657
C04273=1221.093,55.755,-45.177,-178.976,5.505,148.656
C04274=1221.088,56.023,-45.195,-178.973,5.506,148.655
C04275=1221.082,56.273,-45.212,-178.971,5.507,148.655
C04276=1221.078,56.522,-45.229,-178.968,5.508,148.654
C04277=1221.073,56.772,-45.246,-178.966,5.508,148.654
C04278=1221.067,57.021,-45.262,-178.963,5.509,148.653
C04279=1221.063,57.271,-45.278,-178.960,5.509,148.652
C04280=1221.058,57.520,-45.295,-178.958,5.510,148.652
C04281=1221.053,57.769,-45.312,-178.956,5.511,148.651
C04282=1221.048,58.019,-45.329,-178.953,5.512,148.650
C04283=1221.044,58.268,-45.345,-178.950,5.512,148.650
C04284=1221.038,58.518,-45.362,-178.948,5.513,148.649
C04285=1221.034,58.766,-45.380,-178.945,5.513,148.648
C04286=1221.029,59.016,-45.396,-178.943,5.514,148.648
C04287=1221.024,59.266,-45.414,-178.940,5.515,148.647
C04288=1221.019,59.514,-45.430,-178.938,5.515,148.647
C04289=1221.014,59.764,-45.447,-178.935,5.516,148.646
C04290=1221.009,60.014,-45.464,-178.932,5.516,148.645
C04291=1221.004,60.264,-45.481,-178.930,5.517,148.645
C04292=1220.999,60.512,-45.497,-178.928,5.518,148.644
C04293=1220.994,60.762,-45.514,-178.925,5.518,148.644
C04294=1220.989,61.012,-45.531,-178.922,5.519,148.643
C04295=1220.985,61.261,-45.548,-178.920,5.520,148.642
C04296=1220.979,61.510,-45.565,-178.918,5.521,148.642
C04297=1220.975,61.759,-45.582,-178.915,5.521,148.641
C04298=1220.969,62.009,-45.599,-178.912,5.522,148.640
C04299=1220.965,62.258,-45.616,-178.910,5.522,148.640
C04300=1220.959,62.507,-45.633,-178.907,5.523,148.639
C04301=1220.955,62.757,-45.650,-178.905,5.524,148.639
C04302=1220.950,63.006,-45.666,-178.902,5.524,148.638
C04303=1220.945,63.256,-45.684,-178.900,5.525,148.637
C04304=1220.941,63.505,-45.701,-178.897,5.525,148.637
C04305=1220.935,63.754,-45.718,-178.894,5.526,148.636
C04306=1220.930,64.004,-45.735,-178.892,5.527,148.636
C04307=1220.925,64.253,-45.752,-178.890,5.528,148.635
C04308=1220.921,64.502,-45.769,-178.887,5.528,148.634
C04309=1220.916,64.752,-45.787,-178.884,5.529,148.634
C04310=1220.910,65.001,-45.803,-178.882,5.529,148.633
C04311=1220.906,65.251,-45.820,-178.880,5.530,148.633
C04312=1220.901,65.500,-45.838,-178.876,5.532,148.632
C04313=1220.896,65.749,-45.855,-178.874,5.532,148.631
C04314=1220.891,65.999,-45.872,-178.871,5.533,148.631
C04315=1220.886,66.249,-45.889,-178.869,5.534,148.630
C04316=1220.881,66.497,-45.906,-178.866,5.534,148.629
C04317=1220.876,66.747,-45.923,-178.864,5.535,148.629
C04318=1220.871,66.996,-45.940,-178.861,5.535,148.628
C04319=1220.866,67.245,-45.958,-178.858,5.536,148.627
C04320=1220.862,67.495,-45.975,-178.856,5.537,148.627
C04321=1220.857,67.745,-45.992,-178.854,5.537,148.626
C04322=1220.852,67.993,-46.009,-178.851,5.538,148.626
C04323=1220.847,68.243,-46.026,-178.848,5.539,148.625
C04324=1220.842,68.492,-46.043,-178.846,5.540,148.625
C04325=1220.837,68.741,-46.061,-178.844,5.540,148.624
C04326=1220.832,68.991,-46.078,-178.841,5.541,148.623
C04327=1220.828,69.240,-46.096,-178.838,5.541,148.623
C04328=1220.823,69.490,-46.113,-178.836,5.542,148.622
C04329=1220.817,69.740,-46.130,-178.833,5.544,148.622
C04330=1220.813,69.989,-46.148,-178.830,5.544,148.621
C04331=1220.807,70.238,-46.165,-178.828,5.545,148.620
C04332=1220.803,70.487,-46.182,-178.825,5.545,148.620
C04333=1220.798,70.736,-46.199,-178.823,5.546,148.619
C04334=1220.793,70.985,-46.217,-178.820,5.547,148.618
C04335=1220.788,71.235,-46.234,-178.818,5.547,148.618
C04336=1220.784,71.484,-46.252,-178.815,5.548,148.617
C04337=1220.779,71.734,-46.269,-178.813,5.549,148.617
C04338=1220.774,71.983,-46.287,-178.810,5.549,148.616
C04339=1220.769,72.233,-46.304,-178.808,5.550,148.615
C04340=1220.764,72.482,-46.322,-178.805,5.551,148.615
C04341=1220.759,72.732,-46.339,-178.803,5.552,148.614
C04342=1220.754,72.981,-46.357,-178.800,5.553,148.614
C04343=1220.750,73.230,-46.374,-178.797,5.554,148.613
C04344=1220.744,73.479,-46.391,-178.795,5.554,148.612
C04345=1220.739,73.728,-46.408,-178.792,5.555,148.612
C04346=1220.735,73.977,-46.426,-178.790,5.556,148.611
C04347=1220.730,74.227,-46.443,-178.787,5.556,148.611
C04348=1220.725,74.476,-46.461,-178.785,5.557,148.610
C04349=1220.719,74.726,-46.478,-178.782,5.557,148.609
C04350=1220.715,74.975,-46.496,-178.780,5.558,148.609
C04351=1220.710,75.224,-46.514,-178.777,5.559,148.608
C04352=1220.705,75.474,-46.531,-178.775,5.559,148.608
C04353=1220.700,75.723,-46.549,-178.771,5.561,148.607
C04354=1220.695,75.972,-46.567,-178.769,5.562,148.606
C04355=1220.691,76.222,-46.584,-178.767,5.562,148.606
C04356=1220.686,76.471,-46.602,-178.764,5.563,148.605
C04357=1220.681,76.721,-46.619,-178.762,5.564,148.605
C04358=1220.676,76.970,-46.637,-178.759,5.565,148.604
C04359=1220.671,77.219,-46.655,-178.757,5.565,148.603
C04360=1220.666,77.469,-46.672,-178.754,5.566,148.603
C04361=1220.661,77.718,-46.689,-178.752,5.567,148.602
C04362=1220.657,77.967,-46.707,-178.749,5.568,148.602
C04363=1220.652,78.216,-46.725,-178.746,5.569,148.601
C04364=1220.646,78.466,-46.743,-178.743,5.569,148.600
C04365=1220.641,78.715,-46.761,-178.741,5.570,148.600
C04366=1220.637,78.964,-46.779,-178.739,5.571,148.599
C04367=1220.632,79.214,-46.795,-178.736,5.571,148.599
C04368=1220.627,79.463,-46.813,-178.733,5.572,148.598
C04369=1220.622,79.712,-46.831,-178.731,5.573,148.597
C04370=1220.617,79.961,-46.849,-178.729,5.573,148.597
C04371=1220.613,80.211,-46.868,-178.725,5.575,148.596
C04372=1220.608,80.461,-46.885,-178.723,5.576,148.596
C04373=1220.603,80.710,-46.903,-178.721,5.576,148.595
C04374=1220.598,80.959,-46.921,-178.718,5.577,148.594
C04375=1220.593,81.228,-46.940,-178.715,5.577,148.594
C04376=1220.588,81.496,-46.959,-178.712,5.579,148.593
C04377=1220.582,81.764,-46.978,-178.710,5.579,148.593
C04378=1220.577,82.032,-46.997,-178.707,5.580,148.592
C04379=1220.572,82.281,-47.015,-178.705,5.581,148.591
C04380=1220.568,82.531,-47.034,-178.702,5.582,148.591
C04381=1220.562,82.781,-47.051,-178.699,5.583,148.590
C04382=1220.557,83.030,-47.069,-178.697,5.584,148.590
C04383=1220.552,83.279,-47.087,-178.694,5.585,148.589
C04384=1220.548,83.529,-47.105,-178.692,5.585,148.588
C04385=1220.543,83.778,-47.123,-178.689,5.586,148.588
C04386=1220.538,84.027,-47.141,-178.687,5.587,148.587
C04387=1220.533,84.276,-47.159,-178.684,5.587,148.587
C04388=1220.528,84.525,-47.177,-178.681,5.589,148.586
C04389=1220.524,84.775,-47.195,-178.679,5.590,148.586
C04390=1220.519,85.024,-47.213,-178.676,5.590,148.585
C04391=1220.514,85.274,-47.231,-178.674,5.591,148.584
C04392=1220.509,85.523,-47.249,-178.671,5.591,148.584
C04393=1220.504,85.772,-47.266,-178.669,5.592,148.583
C04394=1220.499,86.022,-47.284,-178.666,5.593,148.583
C04395=1220.494,86.271,-47.302,-178.663,5.594,148.582
C04396=1220.490,86.521,-47.321,-178.661,5.595,148.581
C04397=1220.485,86.770,-47.339,-178.658,5.596,148.581
C04398=1220.480,87.018,-47.357,-178.656,5.596,148.580
C04399=1220.475,87.268,-47.375,-178.654,5.597,148.580
C04400=1220.470,87.517,-47.393,-178.651,5.598,148.579
C04401=1220.465,87.766,-47.411,-178.648,5.599,148.578
C04402=1220.461,88.016,-47.430,-178.646,5.600,148.578
C04403=1220.456,88.265,-47.448,-178.643,5.601,148.577
C04404=1220.450,88.514,-47.466,-178.640,5.601,148.577
C04405=1220.445,88.764,-47.484,-178.638,5.602,148.576
C04406=1220.441,89.013,-47.502,-178.636,5.603,148.576
C04407=1220.436,89.263,-47.521,-178.632,5.604,148.575
C04408=1220.431,89.512,-47.538,-178.630,5.605,148.574
C04409=1220.426,89.761,-47.556,-178.628,5.606,148.574
C04410=1220.422,90.010,-47.574,-178.625,5.607,148.573
C04411=1220.417,90.259,-47.593,-178.622,5.607,148.573
C04412=1220.412,90.509,-47.612,-178.620,5.608,148.572
C04413=1220.407,90.758,-47.630,-178.617,5.610,148.572
C04414=1220.402,91.007,-47.648,-178.614,5.610,148.571
C04415=1220.397,91.257,-47.666,-178.612,5.611,148.570
C04416=1220.392,91.506,-47.684,-178.610,5.612,148.570
C04417=1220.388,91.755,-47.703,-178.607,5.612,148.569
C04418=1220.383,92.004,-47.722,-178.605,5.613,148.569
C04419=1220.378,92.254,-47.740,-178.602,5.615,148.568
C04420=1220.373,92.503,-47.758,-178.599,5.615,148.567
C04421=1220.368,92.753,-47.776,-178.597,5.616,148.567
C04422=1220.364,93.001,-47.795,-178.594,5.617,148.566
C04423=1220.358,93.251,-47.813,-178.592,5.617,148.566
C04424=1220.353,93.500,-47.831,-178.589,5.619,148.565
C04425=1220.349,93.750,-47.850,-178.586,5.620,148.565
C04426=1220.344,93.998,-47.868,-178.584,5.620,148.564
C04427=1220.339,94.248,-47.887,-178.582,5.621,148.564
C04428=1220.334,94.498,-47.905,-178.579,5.622,148.563
C04429=1220.330,94.746,-47.924,-178.576,5.623,148.562
C04430=1220.325,94.995,-47.942,-178.574,5.624,148.562
C04431=1220.319,95.245,-47.960,-178.571,5.625,148.561
C04432=1220.315,95.495,-47.979,-178.569,5.625,148.561
C04433=1220.310,95.743,-47.997,-178.566,5.626,148.560
C04434=1220.305,95.993,-48.016,-178.563,5.628,148.560
C04435=1220.301,96.242,-48.035,-178.561,5.628,148.559
C04436=1220.296,96.491,-48.053,-178.558,5.629,148.558
C04437=1220.291,96.740,-48.071,-178.556,5.630,148.558
C04438=1220.286,96.990,-48.091,-178.553,5.631,148.557
C04439=1220.281,97.239,-48.109,-178.551,5.632,148.557
C04440=1220.276,97.488,-48.127,-178.548,5.633,148.556
C04441=1220.272,97.738,-48.146,-178.545,5.633,148.555
C04442=1220.267,97.987,-48.164,-178.543,5.634,148.555
C04443=1220.262,98.236,-48.183,-178.540,5.636,148.554
C04444=1220.257,98.486,-48.202,-178.538,5.637,148.554
C04445=1220.252,98.734,-48.221,-178.535,5.637,148.553
C04446=1220.247,98.984,-48.239,-178.533,5.638,148.553
C04447=1220.242,99.234,-48.258,-178.531,5.639,148.552
C04448=1220.238,99.482,-48.276,-178.527,5.640,148.552
C04449=1220.232,99.732,-48.295,-178.525,5.641,148.551
C04450=1220.228,99.981,-48.314,-178.523,5.642,148.551
C04451=1220.223,100.230,-48.332,-178.520,5.643,148.550
C04452=1220.218,100.480,-48.352,-178.517,5.644,148.549
C04453=1220.214,100.729,-48.370,-178.515,5.645,148.549
C04454=1220.208,100.978,-48.389,-178.512,5.646,148.548
C04455=1220.204,101.228,-48.407,-178.510,5.646,148.548
C04456=1220.199,101.476,-48.426,-178.507,5.648,148.547
C04457=1220.194,101.725,-48.445,-178.504,5.649,148.547
C04458=1220.190,101.975,-48.463,-178.502,5.649,148.546
C04459=1220.184,102.224,-48.483,-178.499,5.650,148.545
C04460=1220.180,102.474,-48.501,-178.496,5.651,148.545
C04461=1220.175,102.723,-48.520,-178.494,5.652,148.544
C04462=1220.170,102.973,-48.539,-178.491,5.653,148.544
C04463=1220.165,103.221,-48.558,-178.489,5.654,148.543
C04464=1220.160,103.470,-48.577,-178.487,5.655,148.543
C04465=1220.155,103.720,-48.596,-178.484,5.656,148.542
C04466=1220.151,103.969,-48.614,-178.481,5.657,148.542
C04467=1220.146,104.218,-48.634,-178.479,5.658,148.541
C04468=1220.141,104.467,-48.652,-178.477,5.659,148.541
C04469=1220.136,104.717,-48.672,-178.473,5.660,148.540
C04470=1220.132,104.966,-48.690,-178.471,5.661,148.539
C04471=1220.126,105.215,-48.709,-178.469,5.662,148.539
C04472=1220.122,105.464,-48.728,-178.466,5.663,148.538
C04473=1220.117,105.713,-48.747,-178.463,5.664,148.538
C04474=1220.112,105.963,-48.766,-178.461,5.665,148.537
C04475=1220.107,106.212,-48.785,-178.458,5.665,148.537
C04476=1220.103,106.461,-48.804,-178.456,5.667,148.536
C04477=1220.097,106.711,-48.823,-178.453,5.668,148.536
C04478=1220.093,106.960,-48.842,-178.450,5.668,148.535
C04479=1220.088,107.228,-48.862,-178.448,5.670,148.534
C04480=1220.083,107.497,-48.883,-178.445,5.670,148.534
C04481=1220.077,107.765,-48.903,-178.442,5.671,148.533
C04482=1220.072,108.034,-48.925,-178.439,5.673,148.533
C04483=1220.068,108.282,-48.943,-178.437,5.673,148.532
C04484=1220.063,108.532,-48.962,-178.434,5.674,148.531
C04485=1220.058,108.781,-48.981,-178.432,5.676,148.531
C04486=1220.053,109.031,-49.001,-178.429,5.676,148.530
C04487=1220.048,109.279,-49.020,-178.427,5.677,148.530
C04488=1220.044,109.529,-49.039,-178.424,5.679,148.529
C04489=1220.039,109.778,-49.058,-178.421,5.679,148.529
C04490=1220.033,110.028,-49.077,-178.419,5.680,148.528
C04491=1220.029,110.276,-49.096,-178.416,5.681,148.528
C04492=1220.024,110.526,-49.115,-178.413,5.682,148.527
C04493=1220.019,110.775,-49.135,-178.411,5.683,148.527
C04494=1220.015,111.024,-49.154,-178.409,5.684,148.526
C04495=1220.010,111.274,-49.173,-178.406,5.686,148.526
C04496=1220.005,111.522,-49.193,-178.403,5.686,148.525
C04497=1220.001,111.772,-49.212,-178.401,5.687,148.525
C04498=1219.995,112.021,-49.231,-178.399,5.688,148.524
C04499=1219.991,112.270,-49.251,-178.395,5.689,148.523
C04500=1219.986,112.519,-49.269,-178.393,5.690,148.523
C04501=1219.981,112.769,-49.288,-178.391,5.691,148.522
C04502=1219.976,113.018,-49.308,-178.388,5.693,148.522
C04503=1219.971,113.267,-49.327,-178.385,5.693,148.521
C04504=1219.967,113.517,-49.346,-178.383,5.694,148.521
C04505=1219.962,113.765,-49.366,-178.380,5.696,148.520
C04506=1219.957,114.015,-49.385,-178.377,5.696,148.520
C04507=1219.951,114.264,-49.405,-178.375,5.697,148.519
C04508=1219.947,114.513,-49.424,-178.372,5.699,148.518
C04509=1219.943,114.763,-49.443,-178.370,5.700,148.518
C04510=1219.937,115.012,-49.463,-178.367,5.700,148.517
C04511=1219.933,115.261,-49.483,-178.365,5.701,148.517
C04512=1219.929,115.510,-49.502,-178.362,5.703,148.516
C04513=1219.924,115.759,-49.521,-178.360,5.704,148.516
C04514=1219.919,116.008,-49.541,-178.357,5.704,148.515
C04515=1219.913,116.257,-49.560,-178.354,5.706,148.515
C04516=1219.909,116.507,-49.580,-178.352,5.707,148.514
C04517=1219.905,116.756,-49.599,-178.349,5.707,148.514
C04518=1219.899,117.005,-49.618,-178.347,5.709,148.513
C04519=1219.895,117.254,-49.638,-178.344,5.710,148.513
C04520=1219.890,117.504,-49.658,-178.342,5.711,148.512
C04521=1219.885,117.752,-49.678,-178.339,5.712,148.512
C04522=1219.880,118.002,-49.697,-178.337,5.713,148.511
C04523=1219.876,118.251,-49.716,-178.334,5.714,148.511
C04524=1219.871,118.500,-49.736,-178.331,5.716,148.510
C04525=1219.866,118.749,-49.755,-178.329,5.716,148.510
C04526=1219.861,118.999,-49.775,-178.326,5.717,148.509
C04527=1219.856,119.247,-49.795,-178.324,5.719,148.508
C04528=1219.852,119.497,-49.815,-178.321,5.719,148.508
C04529=1219.847,119.746,-49.834,-178.319,5.720,148.507
C04530=1219.841,119.995,-49.854,-178.316,5.722,148.507
C04531=1219.837,120.244,-49.874,-178.314,5.723,148.506
C04532=1219.833,120.493,-49.893,-178.311,5.723,148.506
C04533=1219.828,120.742,-49.912,-178.308,5.725,148.505
C04534=1219.823,120.992,-49.932,-178.306,5.726,148.505
C04535=1219.818,121.241,-49.952,-178.304,5.727,148.504
C04536=1219.814,121.490,-49.972,-178.300,5.728,148.504
C04537=1219.808,121.739,-49.991,-178.298,5.729,148.503
C04538=1219.804,121.989,-50.011,-178.295,5.730,148.503
C04539=1219.799,122.238,-50.031,-178.293,5.731,148.502
C04540=1219.794,122.487,-50.051,-178.290,5.732,148.502
C04541=1219.789,122.736,-50.070,-178.288,5.734,148.501
C04542=1219.785,122.985,-50.091,-178.285,5.734,148.501
C04543=1219.780,123.235,-50.110,-178.283,5.735,148.500
C04544=1219.775,123.484,-50.130,-178.280,5.737,148.500
C04545=1219.770,123.733,-50.150,-178.277,5.737,148.499
C04546=1219.765,123.982,-50.170,-178.275,5.738,148.499
C04547=1219.761,124.231,-50.190,-178.272,5.740,148.498
C04548=1219.756,124.481,-50.210,-178.270,5.741,148.498
C04549=1219.751,124.730,-50.229,-178.267,5.742,148.497
C04550=1219.746,124.978,-50.249,-178.264,5.743,148.496
C04551=1219.742,125.228,-50.269,-178.262,5.744,148.496
C04552=1219.737,125.477,-50.289,-178.259,5.746,148.495
C04553=1219.733,125.727,-50.309,-178.257,5.746,148.495
C04554=1219.727,125.975,-50.329,-178.254,5.747,148.494
C04555=1219.723,126.224,-50.349,-178.251,5.749,148.494
C04556=1219.718,126.473,-50.369,-178.249,5.750,148.493
C04557=1219.714,126.723,-50.389,-178.246,5.751,148.493
C04558=1219.709,126.972,-50.409,-178.244,5.752,148.492
C04559=1219.703,127.221,-50.429,-178.241,5.753,148.492
C04560=1219.699,127.470,-50.449,-178.239,5.754,148.491
C04561=1219.694,127.720,-50.469,-178.236,5.755,148.491
C04562=1219.689,127.968,-50.489,-178.233,5.757,148.490
C04563=1219.685,128.218,-50.509,-178.231,5.758,148.490
C04564=1219.680,128.467,-50.529,-178.229,5.758,148.489
C04565=1219.675,128.716,-50.549,-178.226,5.760,148.489
C04566=1219.670,128.965,-50.569,-178.223,5.761,148.488
C04567=1219.666,129.214,-50.589,-178.221,5.762,148.488
C04568=1219.661,129.464,-50.610,-178.218,5.763,148.487
C04569=1219.656,129.713,-50.630,-178.216,5.764,148.487
C04570=1219.651,129.962,-50.650,-178.213,5.766,148.486
C04571=1219.646,130.210,-50.670,-178.211,5.767,148.486
C04572=1219.642,130.460,-50.689,-178.208,5.767,148.485
C04573=1219.637,130.709,-50.710,-178.205,5.769,148.485
C04574=1219.632,130.958,-50.731,-178.203,5.770,148.484
C04575=1219.627,131.208,-50.750,-178.200,5.772,148.484
C04576=1219.623,131.457,-50.771,-178.197,5.772,148.483
C04577=1219.618,131.706,-50.791,-178.195,5.774,148.483
C04578=1219.614,131.955,-50.811,-178.192,5.775,148.482
C04579=1219.608,132.204,-50.832,-178.190,5.776,148.482
C04580=1219.603,132.453,-50.852,-178.187,5.777,148.481
C04581=1219.599,132.702,-50.872,-178.185,5.778,148.481
C04582=1219.594,132.951,-50.892,-178.182,5.780,148.480
C04583=1219.589,133.220,-50.914,-178.179,5.780,148.480
C04584=1219.584,133.489,-50.936,-178.176,5.782,148.479
C04585=1219.579,133.757,-50.958,-178.174,5.783,148.479
C04586=1219.574,134.026,-50.980,-178.171,5.784,148.478
C04587=1219.569,134.275,-51.000,-178.168,5.786,148.477
C04588=1219.565,134.524,-51.020,-178.166,5.787,148.477
C04589=1219.559,134.773,-51.041,-178.164,5.788,148.477
C04590=1219.555,135.023,-51.061,-178.160,5.789,148.476
C04591=1219.550,135.272,-51.081,-178.158,5.790,148.476
C04592=1219.545,135.521,-51.102,-178.155,5.792,148.475
C04593=1219.541,135.770,-51.123,-178.153,5.793,148.475
C04594=1219.536,136.019,-51.143,-178.150,5.794,148.474
C04595=1219.530,136.268,-51.164,-178.148,5.795,148.474
C04596=1219.526,136.517,-51.183,-178.145,5.796,148.473
C04597=1219.521,136.766,-51.204,-178.143,5.797,148.473
C04598=1219.516,137.015,-51.225,-178.140,5.798,148.472
C04599=1219.512,137.264,-51.245,-178.137,5.800,148.472
C04600=1219.507,137.513,-51.265,-178.135,5.801,148.471
C04601=1219.502,137.763,-51.286,-178.132,5.802,148.471
C04602=1219.498,138.011,-51.307,-178.130,5.803,148.470
C04603=1219.493,138.260,-51.327,-178.127,5.805,148.470
C04604=1219.488,138.510,-51.348,-178.125,5.806,148.469
C04605=1219.484,138.759,-51.368,-178.122,5.807,148.469
C04606=1219.478,139.008,-51.389,-178.119,5.808,148.468
C04607=1219.474,139.257,-51.410,-178.117,5.809,148.468
C04608=1219.470,139.506,-51.430,-178.114,5.811,148.467
C04609=1219.464,139.755,-51.451,-178.112,5.811,148.467
C04610=1219.460,140.004,-51.472,-178.109,5.813,148.466
C04611=1219.455,140.253,-51.492,-178.107,5.814,148.466
C04612=1219.451,140.503,-51.513,-178.104,5.816,148.465
C04613=1219.446,140.752,-51.534,-178.101,5.816,148.465
C04614=1219.441,141.001,-51.555,-178.099,5.818,148.464
C04615=1219.437,141.250,-51.575,-178.096,5.819,148.464
C04616=1219.432,141.499,-51.596,-178.093,5.821,148.463
C04617=1219.427,141.748,-51.616,-178.091,5.822,148.463
C04618=1219.422,141.998,-51.637,-178.088,5.823,148.462
C04619=1219.418,142.247,-51.658,-178.086,5.824,148.462
C04620=1219.412,142.496,-51.679,-178.083,5.825,148.461
C04621=1219.408,142.745,-51.699,-178.081,5.826,148.461
C04622=1219.403,142.994,-51.720,-178.079,5.827,148.461
C04623=1219.398,143.243,-51.740,-178.076,5.829,148.460
C04624=1219.393,143.492,-51.761,-178.073,5.830,148.460
C04625=1219.389,143.741,-51.782,-178.070,5.831,148.459
C04626=1219.385,143.990,-51.804,-178.068,5.832,148.459
C04627=1219.380,144.239,-51.824,-178.065,5.834,148.458
C04628=1219.375,144.489,-51.845,-178.063,5.835,148.457
C04629=1219.370,144.738,-51.866,-178.060,5.837,148.457
C04630=1219.365,144.987,-51.886,-178.058,5.837,148.456
C04631=1219.360,145.236,-51.908,-178.055,5.839,148.456
C04632=1219.356,145.484,-51.928,-178.053,5.840,148.456
C04633=1219.351,145.734,-51.949,-178.050,5.841,148.455
C04634=1219.346,145.983,-51.970,-178.048,5.842,148.455
C04635=1219.342,146.232,-51.992,-178.044,5.844,148.454
C04636=1219.337,146.481,-52.013,-178.042,5.845,148.454
C04637=1219.333,146.730,-52.033,-178.040,5.847,148.453
C04638=1219.327,146.980,-52.054,-178.037,5.847,148.453
C04639=1219.323,147.228,-52.075,-178.034,5.849,148.452
C04640=1219.318,147.477,-52.096,-178.032,5.850,148.452
C04641=1219.313,147.726,-52.117,-178.029,5.852,148.451
C04642=1219.309,147.975,-52.139,-178.027,5.853,148.451
C04643=1219.304,148.225,-52.160,-178.024,5.854,148.450
C04644=1219.299,148.474,-52.181,-178.022,5.855,148.450
C04645=1219.295,148.722,-52.202,-178.019,5.857,148.450
C04646=1219.290,148.971,-52.223,-178.016,5.857,148.449
C04647=1219.285,149.221,-52.244,-178.014,5.859,148.449
C04648=1219.281,149.470,-52.265,-178.012,5.860,148.448
C04649=1219.276,149.719,-52.286,-178.009,5.862,148.448
C04650=1219.271,149.968,-52.307,-178.006,5.863,148.447
C04651=1219.267,150.217,-52.328,-178.004,5.864,148.447
C04652=1219.261,150.466,-52.349,-178.001,5.866,148.446
C04653=1219.257,150.715,-52.371,-177.998,5.867,148.446
C04654=1219.253,150.964,-52.391,-177.995,5.868,148.445
C04655=1219.247,151.213,-52.412,-177.993,5.869,148.445
C04656=1219.243,151.462,-52.434,-177.991,5.871,148.444
C04657=1219.238,151.712,-52.455,-177.988,5.872,148.444
C04658=1219.234,151.960,-52.476,-177.985,5.874,148.443
C04659=1219.229,152.210,-52.497,-177.983,5.875,148.443
C04660=1219.224,152.458,-52.519,-177.980,5.876,148.442
C04661=1219.219,152.708,-52.540,-177.978,5.877,148.442
C04662=1219.215,152.957,-52.562,-177.975,5.879,148.442
C04663=1219.210,153.206,-52.582,-177.973,5.880,148.441
C04664=1219.205,153.454,-52.604,-177.970,5.881,148.441
C04665=1219.200,153.704,-52.625,-177.967,5.883,148.440
C04666=1219.196,153.953,-52.647,-177.965,5.884,148.440
C04667=1219.191,154.202,-52.668,-177.962,5.886,148.439
C04668=1219.186,154.451,-52.689,-177.960,5.887,148.439
C04669=1219.182,154.700,-52.711,-177.957,5.888,148.438
C04670=1219.177,154.949,-52.732,-177.955,5.889,148.438
C04671=1219.172,155.198,-52.754,-177.952,5.891,148.438
C04672=1219.167,155.447,-52.775,-177.949,5.891,148.437
C04673=1219.163,155.696,-52.796,-177.947,5.893,148.437
C04674=1219.158,155.945,-52.818,-177.944,5.895,148.436
C04675=1219.153,156.194,-52.839,-177.942,5.896,148.436
C04676=1219.149,156.443,-52.861,-177.939,5.898,148.435
C04677=1219.144,156.692,-52.883,-177.937,5.899,148.435
C04678=1219.139,156.941,-52.904,-177.934,5.900,148.434
C04679=1219.135,157.191,-52.926,-177.932,5.901,148.434
C04680=1219.130,157.439,-52.947,-177.929,5.903,148.433
C04681=1219.125,157.688,-52.968,-177.926,5.904,148.433
C04682=1219.121,157.938,-52.990,-177.924,5.905,148.432
C04683=1219.116,158.186,-53.012,-177.921,5.907,148.432
C04684=1219.111,158.435,-53.033,-177.918,5.908,148.431
C04685=1219.107,158.685,-53.055,-177.916,5.910,148.431
C04686=1219.102,158.933,-53.076,-177.914,5.911,148.431
C04687=1219.096,159.203,-53.100,-177.910,5.912,148.430
C04688=1219.092,159.472,-53.122,-177.908,5.914,148.430
C04689=1219.087,159.741,-53.146,-177.905,5.915,148.429
C04690=1219.082,160.010,-53.169,-177.902,5.917,148.429
C04691=1219.077,160.258,-53.191,-177.900,5.918,148.428
C04692=1219.073,160.508,-53.213,-177.897,5.920,148.428
C04693=1219.068,160.756,-53.235,-177.895,5.921,148.427
C04694=1219.063,161.006,-53.256,-177.892,5.922,148.427
C04695=1219.058,161.255,-53.278,-177.889,5.924,148.426
C04696=1219.053,161.504,-53.299,-177.887,5.925,148.426
C04697=1219.049,161.753,-53.321,-177.884,5.927,148.426
C04698=1219.044,162.002,-53.343,-177.882,5.928,148.425
C04699=1219.039,162.250,-53.365,-177.879,5.929,148.425
C04700=1219.035,162.499,-53.387,-177.876,5.931,148.424
C04701=1219.030,162.749,-53.408,-177.874,5.932,148.424
C04702=1219.026,162.998,-53.430,-177.871,5.933,148.423
C04703=1219.021,163.247,-53.451,-177.869,5.934,148.423
C04704=1219.016,163.496,-53.474,-177.866,5.936,148.423
C04705=1219.011,163.745,-53.496,-177.863,5.938,148.422
C04706=1219.006,163.994,-53.517,-177.861,5.939,148.422
C04707=1219.002,164.243,-53.540,-177.858,5.941,148.421
C04708=1218.997,164.492,-53.561,-177.856,5.941,148.421
C04709=1218.993,164.741,-53.583,-177.853,5.943,148.420
C04710=1218.988,164.990,-53.605,-177.850,5.945,148.420
C04711=1218.984,165.239,-53.627,-177.848,5.946,148.420
C04712=1218.979,165.488,-53.649,-177.845,5.948,148.419
C04713=1218.974,165.737,-53.671,-177.842,5.949,148.419
C04714=1218.970,165.986,-53.692,-177.840,5.950,148.418
C04715=1218.965,166.235,-53.715,-177.838,5.952,148.418
C04716=1218.960,166.484,-53.737,-177.835,5.953,148.417
C04717=1218.955,166.733,-53.759,-177.832,5.954,148.417
C04718=1218.951,166.982,-53.780,-177.830,5.956,148.416
C04719=1218.946,167.231,-53.803,-177.828,5.957,148.416
C04720=1218.941,167.480,-53.824,-177.825,5.959,148.416
C04721=1218.937,167.729,-53.847,-177.822,5.960,148.415
C04722=1218.932,167.978,-53.869,-177.820,5.961,148.415
C04723=1218.928,168.227,-53.891,-177.817,5.963,148.414
C04724=1218.923,168.475,-53.913,-177.815,5.964,148.414
C04725=1218.918,168.725,-53.935,-177.812,5.966,148.413
C04726=1218.914,168.973,-53.957,-177.809,5.968,148.413
C04727=1218.909,169.223,-53.979,-177.807,5.969,148.413
C04728=1218.904,169.471,-54.002,-177.804,5.970,148.412
C04729=1218.900,169.720,-54.024,-177.801,5.972,148.412
C04730=1218.895,169.969,-54.045,-177.799,5.973,148.411
C04731=1218.890,170.219,-54.068,-177.796,5.975,148.411
C04732=1218.885,170.467,-54.090,-177.794,5.977,148.411
C04733=1218.881,170.716,-54.113,-177.791,5.977,148.410
C04734=1218.876,170.965,-54.134,-177.789,5.979,148.410
C04735=1218.871,171.214,-54.157,-177.786,5.981,148.409
C04736=1218.867,171.464,-54.179,-177.784,5.982,148.409
C04737=1218.862,171.712,-54.201,-177.781,5.983,148.408
C04738=1218.857,171.961,-54.224,-177.778,5.985,148.408
C04739=1218.852,172.210,-54.246,-177.776,5.986,148.408
C04740=1218.848,172.459,-54.268,-177.773,5.988,148.407
C04741=1218.844,172.707,-54.290,-177.771,5.990,148.407
C04742=1218.839,172.957,-54.313,-177.768,5.990,148.406
C04743=1218.834,173.206,-54.335,-177.765,5.992,148.406
C04744=1218.830,173.454,-54.357,-177.763,5.994,148.405
C04745=1218.825,173.704,-54.380,-177.761,5.995,148.405
C04746=1218.820,173.953,-54.402,-177.757,5.997,148.405
C04747=1218.815,174.202,-54.425,-177.755,5.998,148.404
C04748=1218.811,174.451,-54.447,-177.753,5.999,148.404
C04749=1218.806,174.700,-54.469,-177.750,6.001,148.403
C04750=1218.801,174.949,-54.492,-177.747,6.003,148.403
C04751=1218.797,175.198,-54.514,-177.745,6.004,148.402
C04752=1218.793,175.446,-54.536,-177.742,6.005,148.402
C04753=1218.788,175.696,-54.559,-177.739,6.007,148.402
C04754=1218.783,175.944,-54.581,-177.737,6.008,148.401
C04755=1218.778,176.193,-54.604,-177.735,6.010,148.401
C04756=1218.774,176.443,-54.626,-177.732,6.012,148.400
C04757=1218.769,176.691,-54.649,-177.729,6.013,148.400
C04758=1218.764,176.941,-54.671,-177.727,6.014,148.400
C04759=1218.760,177.189,-54.694,-177.724,6.016,148.399
C04760=1218.755,177.438,-54.716,-177.722,6.018,148.399
C04761=1218.751,177.687,-54.739,-177.719,6.019,148.398
C04762=1218.746,177.937,-54.762,-177.716,6.021,148.398
C04763=1218.741,178.185,-54.784,-177.714,6.022,148.398
C04764=1218.736,178.434,-54.807,-177.712,6.023,148.397
C04765=1218.732,178.683,-54.829,-177.709,6.025,148.397
C04766=1218.727,178.931,-54.852,-177.706,6.027,148.396
C04767=1218.723,179.181,-54.874,-177.703,6.029,148.396
C04768=1218.718,179.430,-54.898,-177.701,6.030,148.396
C04769=1218.714,179.679,-54.920,-177.698,6.031,148.395
C04770=1218.708,179.927,-54.943,-177.696,6.033,148.395
C04771=1218.704,180.176,-54.966,-177.694,6.034,148.394
C04772=1218.699,180.426,-54.988,-177.690,6.036,148.394
C04773=1218.695,180.674,-55.011,-177.688,6.038,148.394
C04774=1218.690,180.923,-55.033,-177.685,6.039,148.393
C04775=1218.686,181.172,-55.056,-177.683,6.040,148.393
C04776=1218.681,181.421,-55.079,-177.680,6.042,148.392
C04777=1218.676,181.670,-55.101,-177.678,6.044,148.392
C04778=1218.671,181.919,-55.124,-177.675,6.045,148.391
C04779=1218.668,182.168,-55.147,-177.673,6.047,148.391
C04780=1218.662,182.417,-55.170,-177.670,6.048,148.391
C04781=1218.657,182.666,-55.193,-177.667,6.050,148.390
C04782=1218.653,182.914,-55.216,-177.665,6.051,148.390
C04783=1218.649,183.163,-55.239,-177.662,6.053,148.390
C04784=1218.644,183.413,-55.261,-177.659,6.054,148.389
C04785=1218.640,183.662,-55.284,-177.657,6.056,148.389
C04786=1218.634,183.910,-55.307,-177.655,6.057,148.388
C04787=1218.630,184.159,-55.330,-177.652,6.059,148.388
C04788=1218.625,184.408,-55.353,-177.649,6.061,148.388
C04789=1218.621,184.657,-55.376,-177.647,6.063,148.387
C04790=1218.617,184.906,-55.399,-177.644,6.063,148.387
C04791=1218.611,185.176,-55.424,-177.641,6.065,148.386
C04792=1218.607,185.445,-55.448,-177.639,6.067,148.386
C04793=1218.601,185.715,-55.473,-177.636,6.069,148.386
C04794=1218.596,185.985,-55.498,-177.633,6.070,148.385
C04795=1218.592,186.233,-55.521,-177.630,6.072,148.385
C04796=1218.587,186.482,-55.544,-177.628,6.074,148.384
C04797=1218.582,186.731,-55.568,-177.625,6.076,148.384
C04798=1218.577,186.980,-55.591,-177.623,6.077,148.384
C04799=1218.573,187.229,-55.614,-177.620,6.079,148.383
C04800=1218.569,187.478,-55.637,-177.617,6.080,148.383
C04801=1218.564,187.727,-55.660,-177.615,6.082,148.382
C04802=1218.560,187.975,-55.683,-177.612,6.083,148.382
C04803=1218.555,188.224,-55.706,-177.610,6.085,148.382
C04804=1218.550,188.473,-55.730,-177.607,6.087,148.381
C04805=1218.545,188.722,-55.752,-177.604,6.089,148.381
C04806=1218.541,188.971,-55.775,-177.602,6.090,148.381
C04807=1218.536,189.220,-55.798,-177.600,6.091,148.380
C04808=1218.532,189.469,-55.822,-177.597,6.093,148.380
C04809=1218.526,189.718,-55.845,-177.594,6.095,148.379
C04810=1218.522,189.967,-55.868,-177.591,6.097,148.379
C04811=1218.518,190.215,-55.892,-177.589,6.098,148.379
C04812=1218.513,190.464,-55.915,-177.587,6.099,148.378
C04813=1218.509,190.713,-55.938,-177.584,6.101,148.378
C04814=1218.504,190.962,-55.962,-177.581,6.103,148.378
C04815=1218.499,191.211,-55.985,-177.579,6.104,148.377
C04816=1218.495,191.460,-56.008,-177.577,6.106,148.377
C04817=1218.491,191.709,-56.031,-177.573,6.107,148.376
C04818=1218.486,191.958,-56.054,-177.571,6.109,148.376
C04819=1218.481,192.207,-56.078,-177.568,6.111,148.376
C04820=1218.476,192.455,-56.101,-177.566,6.112,148.375
C04821=1218.471,192.704,-56.124,-177.563,6.114,148.375
C04822=1218.467,192.952,-56.148,-177.561,6.116,148.374
C04823=1218.462,193.201,-56.172,-177.558,6.118,148.374
C04824=1218.457,193.451,-56.195,-177.555,6.120,148.374
C04825=1218.453,193.699,-56.218,-177.553,6.121,148.373
C04826=1218.449,193.948,-56.241,-177.551,6.122,148.373
C04827=1218.444,194.197,-56.264,-177.548,6.124,148.372
C04828=1218.440,194.446,-56.288,-177.545,6.126,148.372
C04829=1218.435,194.695,-56.312,-177.542,6.128,148.372
C04830=1218.430,194.944,-56.335,-177.540,6.129,148.371
C04831=1218.426,195.193,-56.359,-177.538,6.130,148.371
C04832=1218.421,195.441,-56.383,-177.535,6.132,148.371
C04833=1218.416,195.690,-56.406,-177.532,6.134,148.370
C04834=1218.412,195.939,-56.429,-177.530,6.136,148.370
C04835=1218.407,196.188,-56.453,-177.527,6.138,148.370
C04836=1218.403,196.437,-56.477,-177.525,6.139,148.369
C04837=1218.398,196.686,-56.500,-177.522,6.141,148.369
C04838=1218.393,196.935,-56.524,-177.520,6.142,148.369
C04839=1218.389,197.183,-56.548,-177.517,6.144,148.368
C04840=1218.384,197.432,-56.571,-177.514,6.146,148.368
C04841=1218.379,197.681,-56.594,-177.511,6.148,148.367
C04842=1218.375,197.930,-56.618,-177.509,6.149,148.367
C04843=1218.370,198.179,-56.642,-177.506,6.150,148.367
C04844=1218.366,198.428,-56.665,-177.504,6.152,148.366
C04845=1218.361,198.676,-56.689,-177.501,6.154,148.366
C04846=1218.357,198.925,-56.713,-177.499,6.156,148.366
C04847=1218.352,199.174,-56.737,-177.496,6.158,148.365
C04848=1218.348,199.423,-56.760,-177.494,6.159,148.365
C04849=1218.343,199.672,-56.783,-177.491,6.161,148.365
C04850=1218.338,199.920,-56.807,-177.489,6.162,148.364
C04851=1218.334,200.170,-56.831,-177.486,6.164,148.364
C04852=1218.330,200.418,-56.855,-177.483,6.166,148.364
C04853=1218.324,200.668,-56.879,-177.481,6.168,148.363
C04854=1218.320,200.916,-56.903,-177.478,6.170,148.363
C04855=1218.315,201.165,-56.927,-177.476,6.171,148.362
C04856=1218.311,201.413,-56.951,-177.473,6.173,148.362
C04857=1218.306,201.662,-56.974,-177.471,6.175,148.362
C04858=1218.302,201.911,-56.998,-177.468,6.176,148.361
C04859=1218.297,202.160,-57.021,-177.465,6.178,148.361
C04860=1218.293,202.408,-57.046,-177.462,6.180,148.361
C04861=1218.288,202.658,-57.071,-177.460,6.182,148.360
C04862=1218.284,202.907,-57.094,-177.457,6.183,148.360
C04863=1218.279,203.155,-57.118,-177.455,6.184,148.359
C04864=1218.274,203.404,-57.141,-177.452,6.186,148.359
C04865=1218.270,203.653,-57.165,-177.450,6.188,148.359
C04866=1218.265,203.902,-57.189,-177.447,6.190,148.358
C04867=1218.260,204.150,-57.213,-177.444,6.192,148.358
C04868=1218.256,204.399,-57.238,-177.442,6.194,148.358
C04869=1218.252,204.649,-57.261,-177.440,6.195,148.357
C04870=1218.247,204.897,-57.285,-177.437,6.196,148.357
C04871=1218.242,205.146,-57.310,-177.434,6.198,148.357
C04872=1218.238,205.395,-57.333,-177.432,6.200,148.356
C04873=1218.233,205.643,-57.357,-177.429,6.202,148.356
C04874=1218.229,205.892,-57.382,-177.426,6.204,148.356
C04875=1218.224,206.141,-57.407,-177.424,6.206,148.355
C04876=1218.220,206.390,-57.430,-177.421,6.208,148.355
C04877=1218.215,206.638,-57.454,-177.418,6.209,148.355
C04878=1218.211,206.887,-57.478,-177.416,6.210,148.354
C04879=1218.205,207.136,-57.502,-177.414,6.212,148.354
C04880=1218.202,207.385,-57.526,-177.411,6.214,148.354
C04881=1218.197,207.634,-57.551,-177.408,6.216,148.353
C04882=1218.192,207.882,-57.575,-177.406,6.218,148.353
C04883=1218.188,208.131,-57.599,-177.403,6.220,148.353
C04884=1218.183,208.380,-57.623,-177.400,6.221,148.352
C04885=1218.178,208.629,-57.648,-177.398,6.223,148.352
C04886=1218.174,208.878,-57.672,-177.395,6.225,148.352
C04887=1218.170,209.126,-57.696,-177.393,6.227,148.351
C04888=1218.164,209.375,-57.720,-177.390,6.228,148.351
C04889=1218.161,209.624,-57.745,-177.388,6.230,148.351
C04890=1218.156,209.873,-57.768,-177.385,6.232,148.350
C04891=1218.151,210.122,-57.793,-177.383,6.234,148.350
C04892=1218.146,210.370,-57.817,-177.380,6.235,148.350
C04893=1218.142,210.619,-57.841,-177.377,6.237,148.349
C04894=1218.137,210.868,-57.866,-177.375,6.239,148.349
C04895=1218.132,211.138,-57.893,-177.372,6.241,148.349
C04896=1218.128,211.408,-57.919,-177.369,6.243,148.348
C04897=1218.122,211.679,-57.945,-177.366,6.245,148.348
C04898=1218.118,211.950,-57.972,-177.364,6.247,148.348
C04899=1218.113,212.198,-57.997,-177.361,6.249,148.347
C04900=1218.108,212.447,-58.021,-177.358,6.251,148.347
C04901=1218.104,212.695,-58.045,-177.356,6.252,148.347
C04902=1218.099,212.945,-58.070,-177.354,6.254,148.346
C04903=1218.095,213.193,-58.094,-177.351,6.256,148.346
C04904=1218.090,213.442,-58.119,-177.348,6.258,148.346
C04905=1218.086,213.691,-58.143,-177.346,6.259,148.345
C04906=1218.081,213.940,-58.168,-177.343,6.261,148.345
C04907=1218.077,214.188,-58.192,-177.340,6.263,148.345
C04908=1218.072,214.437,-58.217,-177.338,6.265,148.344
C04909=1218.068,214.686,-58.241,-177.335,6.267,148.344
C04910=1218.063,214.935,-58.266,-177.332,6.269,148.344
C04911=1218.059,215.183,-58.291,-177.330,6.271,148.343
C04912=1218.054,215.432,-58.315,-177.327,6.272,148.343
C04913=1218.050,215.680,-58.339,-177.325,6.274,148.343
C04914=1218.045,215.930,-58.365,-177.322,6.276,148.342
C04915=1218.041,216.178,-58.389,-177.319,6.278,148.342
C04916=1218.036,216.427,-58.413,-177.317,6.280,148.342
C04917=1218.031,216.676,-58.438,-177.314,6.282,148.341
C04918=1218.027,216.924,-58.463,-177.311,6.283,148.341
C04919=1218.022,217.173,-58.488,-177.309,6.285,148.341
C04920=1218.018,217.422,-58.512,-177.307,6.287,148.341
C04921=1218.013,217.671,-58.537,-177.305,6.289,148.340
C04922=1218.008,217.920,-58.562,-177.302,6.290,148.340
C04923=1218.004,218.168,-58.587,-177.299,6.292,148.339
C04924=1218.000,218.417,-58.612,-177.297,6.294,148.339
C04925=1217.995,218.666,-58.636,-177.294,6.296,148.339
C04926=1217.990,218.914,-58.660,-177.291,6.298,148.338
C04927=1217.986,219.163,-58.686,-177.289,6.300,148.338
C04928=1217.982,219.412,-58.710,-177.286,6.301,148.338
C04929=1217.977,219.661,-58.735,-177.283,6.303,148.337
C04930=1217.972,219.909,-58.761,-177.281,6.305,148.337
C04931=1217.968,220.157,-58.785,-177.278,6.307,148.337
C04932=1217.963,220.407,-58.810,-177.276,6.309,148.337
C04933=1217.958,220.655,-58.835,-177.273,6.311,148.336
C04934=1217.955,220.904,-58.860,-177.271,6.313,148.336
C04935=1217.949,221.153,-58.884,-177.268,6.315,148.336
C04936=1217.945,221.402,-58.910,-177.266,6.317,148.335
C04937=1217.941,221.650,-58.934,-177.263,6.318,148.335
C04938=1217.937,221.899,-58.960,-177.260,6.320,148.335
C04939=1217.932,222.148,-58.985,-177.258,6.322,148.334
C04940=1217.927,222.397,-59.010,-177.255,6.324,148.334
C04941=1217.923,222.645,-59.034,-177.252,6.326,148.334
C04942=1217.918,222.894,-59.059,-177.250,6.328,148.333
C04943=1217.914,223.142,-59.085,-177.248,6.330,148.333
C04944=1217.908,223.391,-59.109,-177.245,6.332,148.333
C04945=1217.905,223.640,-59.135,-177.242,6.334,148.333
C04946=1217.900,223.888,-59.159,-177.240,6.335,148.332
C04947=1217.896,224.137,-59.185,-177.237,6.337,148.332
C04948=1217.890,224.386,-59.210,-177.234,6.339,148.332
C04949=1217.887,224.634,-59.235,-177.232,6.341,148.331
C04950=1217.882,224.883,-59.260,-177.229,6.343,148.331
C04951=1217.878,225.132,-59.285,-177.227,6.345,148.331
C04952=1217.873,225.381,-59.310,-177.224,6.347,148.331
C04953=1217.868,225.629,-59.336,-177.222,6.349,148.330
C04954=1217.864,225.878,-59.361,-177.219,6.351,148.330
C04955=1217.860,226.127,-59.386,-177.217,6.352,148.330
C04956=1217.855,226.375,-59.411,-177.214,6.354,148.329
C04957=1217.850,226.624,-59.436,-177.211,6.356,148.329
C04958=1217.846,226.873,-59.462,-177.209,6.358,148.329
C04959=1217.841,227.121,-59.487,-177.207,6.360,148.329
C04960=1217.837,227.370,-59.512,-177.204,6.362,148.328
C04961=1217.832,227.619,-59.538,-177.201,6.364,148.328
C04962=1217.828,227.867,-59.563,-177.199,6.366,148.328
C04963=1217.824,228.116,-59.588,-177.196,6.368,148.327
C04964=1217.819,228.365,-59.613,-177.193,6.370,148.327
C04965=1217.815,228.613,-59.639,-177.191,6.372,148.327
C04966=1217.810,228.862,-59.664,-177.189,6.374,148.327
C04967=1217.805,229.111,-59.689,-177.186,6.375,148.326
C04968=1217.801,229.360,-59.715,-177.183,6.377,148.326
C04969=1217.796,229.608,-59.740,-177.181,6.379,148.326
C04970=1217.792,229.857,-59.765,-177.178,6.381,148.325
C04971=1217.787,230.105,-59.791,-177.176,6.383,148.325
C04972=1217.783,230.354,-59.817,-177.173,6.385,148.325
C04973=1217.779,230.603,-59.842,-177.171,6.387,148.325
C04974=1217.773,230.852,-59.867,-177.168,6.389,148.324
C04975=1217.769,231.100,-59.893,-177.165,6.391,148.324
C04976=1217.764,231.349,-59.918,-177.163,6.392,148.324
C04977=1217.760,231.597,-59.944,-177.161,6.395,148.323
C04978=1217.756,231.846,-59.970,-177.158,6.397,148.323
C04979=1217.751,232.094,-59.995,-177.155,6.398,148.323
C04980=1217.747,232.344,-60.020,-177.153,6.400,148.322
C04981=1217.742,232.592,-60.046,-177.150,6.402,148.322
C04982=1217.738,232.841,-60.071,-177.148,6.404,148.322
C04983=1217.733,233.089,-60.097,-177.145,6.406,148.322
C04984=1217.729,233.338,-60.123,-177.143,6.408,148.321
C04985=1217.724,233.586,-60.148,-177.140,6.410,148.321
C04986=1217.720,233.835,-60.174,-177.138,6.412,148.321
C04987=1217.716,234.084,-60.200,-177.135,6.414,148.321
C04988=1217.711,234.332,-60.225,-177.133,6.416,148.320
C04989=1217.707,234.581,-60.251,-177.130,6.418,148.320
C04990=1217.702,234.830,-60.277,-177.127,6.419,148.320
C04991=1217.697,235.078,-60.302,-177.125,6.421,148.319
C04992=1217.693,235.327,-60.328,-177.123,6.424,148.319
C04993=1217.689,235.576,-60.354,-177.120,6.425,148.319
C04994=1217.684,235.824,-60.380,-177.117,6.428,148.319
C04995=1217.679,236.073,-60.405,-177.114,6.430,148.318
C04996=1217.675,236.321,-60.431,-177.112,6.432,148.318
C04997=1217.671,236.570,-60.457,-177.110,6.434,148.318
C04998=1217.666,236.819,-60.483,-177.107,6.436,148.318
C04999=1217.661,237.090,-60.511,-177.104,6.438,148.317
C05000=1217.656,237.362,-60.539,-177.102,6.440,148.317
C05001=1217.651,237.633,-60.567,-177.098,6.442,148.317
C05002=1217.646,237.905,-60.595,-177.096,6.444,148.316
C05003=1217.642,238.154,-60.621,-177.093,6.446,148.316
C05004=1217.637,238.402,-60.646,-177.091,6.448,148.316
C05005=1217.633,238.650,-60.673,-177.088,6.450,148.316
C05006=1217.628,238.899,-60.699,-177.086,6.452,148.315
C05007=1217.624,239.148,-60.725,-177.083,6.454,148.315
C05008=1217.619,239.396,-60.750,-177.081,6.456,148.315
C05009=1217.614,239.645,-60.777,-177.078,6.459,148.315
C05010=1217.611,239.893,-60.803,-177.075,6.461,148.314
C05011=1217.606,240.142,-60.829,-177.073,6.462,148.314
C05012=1217.602,240.391,-60.854,-177.071,6.465,148.314
C05013=1217.597,240.639,-60.880,-177.068,6.466,148.314
C05014=1217.592,240.888,-60.906,-177.065,6.468,148.313
C05015=1217.588,241.136,-60.933,-177.063,6.470,148.313
C05016=1217.584,241.385,-60.958,-177.061,6.472,148.313
C05017=1217.579,241.634,-60.985,-177.058,6.474,148.313
C05018=1217.575,241.882,-61.011,-177.055,6.476,148.312
C05019=1217.570,242.130,-61.037,-177.053,6.478,148.312
C05020=1217.565,242.380,-61.063,-177.051,6.480,148.312
C05021=1217.561,242.628,-61.089,-177.048,6.482,148.312
C05022=1217.557,242.877,-61.115,-177.045,6.485,148.311
C05023=1217.552,243.126,-61.142,-177.042,6.487,148.311
C05024=1217.548,243.374,-61.168,-177.040,6.489,148.311
C05025=1217.544,243.622,-61.193,-177.037,6.491,148.311
C05026=1217.539,243.871,-61.220,-177.035,6.492,148.310
C05027=1217.535,244.119,-61.246,-177.033,6.495,148.310
C05028=1217.530,244.368,-61.273,-177.030,6.497,148.310
C05029=1217.526,244.617,-61.298,-177.027,6.498,148.310
C05030=1217.522,244.865,-61.325,-177.025,6.500,148.309
C05031=1217.517,245.115,-61.351,-177.023,6.502,148.309
C05032=1217.513,245.363,-61.378,-177.020,6.504,148.309
C05033=1217.507,245.611,-61.404,-177.017,6.507,148.309
C05034=1217.503,245.859,-61.430,-177.015,6.509,148.308
C05035=1217.499,246.108,-61.456,-177.012,6.511,148.308
C05036=1217.494,246.357,-61.483,-177.009,6.513,148.308
C05037=1217.490,246.605,-61.509,-177.007,6.515,148.308
C05038=1217.486,246.854,-61.536,-177.005,6.517,148.307
C05039=1217.481,247.103,-61.561,-177.002,6.519,148.307
C05040=1217.477,247.351,-61.588,-176.999,6.521,148.307
C05041=1217.472,247.600,-61.614,-176.997,6.523,148.307
C05042=1217.468,247.849,-61.641,-176.994,6.526,148.306
C05043=1217.464,248.097,-61.667,-176.991,6.527,148.306
C05044=1217.459,248.346,-61.694,-176.989,6.530,148.306
C05045=1217.454,248.593,-61.720,-176.987,6.532,148.306
C05046=1217.449,248.842,-61.747,-176.984,6.533,148.305
C05047=1217.445,249.091,-61.773,-176.982,6.536,148.305
C05048=1217.441,249.340,-61.799,-176.979,6.537,148.305
C05049=1217.437,249.588,-61.826,-176.977,6.539,148.305
C05050=1217.432,249.836,-61.853,-176.974,6.542,148.305
C05051=1217.428,250.085,-61.879,-176.971,6.544,148.304
C05052=1217.423,250.334,-61.906,-176.969,6.546,148.304
C05053=1217.418,250.582,-61.933,-176.967,6.548,148.304
C05054=1217.414,250.831,-61.958,-176.964,6.550,148.304
C05055=1217.410,251.079,-61.986,-176.961,6.552,148.303
C05056=1217.406,251.328,-62.012,-176.959,6.554,148.303
C05057=1217.401,251.576,-62.039,-176.956,6.557,148.303
C05058=1217.396,251.825,-62.065,-176.954,6.559,148.303
C05059=1217.392,252.073,-62.092,-176.951,6.561,148.303
C05060=1217.387,252.322,-62.119,-176.949,6.563,148.302
C05061=1217.383,252.570,-62.145,-176.946,6.565,148.302
C05062=1217.379,252.819,-62.172,-176.944,6.567,148.302
C05063=1217.374,253.068,-62.199,-176.941,6.569,148.302
C05064=1217.370,253.316,-62.225,-176.939,6.572,148.302
C05065=1217.365,253.564,-62.252,-176.936,6.574,148.301
C05066=1217.361,253.813,-62.279,-176.933,6.576,148.301
C05067=1217.357,254.061,-62.306,-176.931,6.578,148.301
C05068=1217.352,254.310,-62.332,-176.929,6.580,148.301
C05069=1217.348,254.559,-62.360,-176.926,6.581,148.300
C05070=1217.344,254.808,-62.386,-176.924,6.584,148.300
C05071=1217.339,255.056,-62.413,-176.921,6.586,148.300
C05072=1217.334,255.305,-62.440,-176.919,6.589,148.300
C05073=1217.330,255.553,-62.467,-176.916,6.590,148.299
C05074=1217.326,255.801,-62.494,-176.913,6.592,148.299
C05075=1217.321,256.050,-62.521,-176.911,6.594,148.299
C05076=1217.317,256.298,-62.548,-176.909,6.596,148.299
C05077=1217.313,256.546,-62.574,-176.906,6.599,148.299
C05078=1217.308,256.795,-62.601,-176.903,6.601,148.298
C05079=1217.303,257.043,-62.628,-176.901,6.603,148.298
C05080=1217.299,257.292,-62.656,-176.899,6.605,148.298
C05081=1217.295,257.541,-62.683,-176.896,6.607,148.298
C05082=1217.291,257.789,-62.709,-176.893,6.610,148.297
C05083=1217.286,258.038,-62.736,-176.891,6.612,148.297
C05084=1217.281,258.286,-62.764,-176.888,6.614,148.297
C05085=1217.277,258.535,-62.791,-176.886,6.616,148.297
C05086=1217.272,258.783,-62.818,-176.883,6.618,148.297
C05087=1217.268,259.031,-62.844,-176.881,6.620,148.297
C05088=1217.264,259.280,-62.871,-176.878,6.623,148.296
C05089=1217.259,259.529,-62.899,-176.875,6.625,148.296
C05090=1217.255,259.778,-62.926,-176.873,6.627,148.296
C05091=1217.250,260.026,-62.953,-176.871,6.629,148.296
C05092=1217.245,260.275,-62.980,-176.869,6.631,148.296
C05093=1217.241,260.523,-63.007,-176.865,6.634,148.295
C05094=1217.237,260.771,-63.034,-176.863,6.636,148.295
C05095=1217.233,261.020,-63.061,-176.861,6.638,148.295
C05096=1217.228,261.268,-63.089,-176.858,6.640,148.295
C05097=1217.224,261.517,-63.116,-176.856,6.642,148.295
C05098=1217.219,261.765,-63.143,-176.853,6.645,148.294
C05099=1217.215,262.013,-63.170,-176.851,6.647,148.294
C05100=1217.210,262.262,-63.198,-176.848,6.649,148.294
C05101=1217.206,262.511,-63.225,-176.846,6.651,148.294
C05102=1217.201,262.759,-63.252,-176.843,6.653,148.294
C05103=1217.197,263.032,-63.282,-176.840,6.655,148.293
C05104=1217.192,263.304,-63.312,-176.837,6.659,148.293
C05105=1217.187,263.577,-63.342,-176.835,6.660,148.293
C05106=1217.182,263.850,-63.372,-176.832,6.663,148.293
C05107=1217.178,264.099,-63.399,-176.830,6.665,148.293
C05108=1217.173,264.347,-63.427,-176.827,6.667,148.292
C05109=1217.169,264.595,-63.454,-176.825,6.669,148.292
C05110=1217.165,264.844,-63.482,-176.822,6.672,148.292
C05111=1217.160,265.093,-63.509,-176.819,6.674,148.292
C05112=1217.156,265.340,-63.537,-176.817,6.676,148.292
C05113=1217.151,265.589,-63.564,-176.815,6.678,148.291
C05114=1217.147,265.838,-63.591,-176.812,6.680,148.291
C05115=1217.143,266.086,-63.619,-176.809,6.683,148.291
C05116=1217.138,266.335,-63.646,-176.807,6.685,148.291
C05117=1217.134,266.582,-63.674,-176.804,6.687,148.291
C05118=1217.130,266.832,-63.701,-176.802,6.689,148.290
C05119=1217.125,267.080,-63.728,-176.799,6.692,148.290
C05120=1217.121,267.328,-63.756,-176.797,6.694,148.290
C05121=1217.116,267.576,-63.783,-176.794,6.696,148.290
C05122=1217.112,267.825,-63.811,-176.792,6.698,148.290
C05123=1217.108,268.074,-63.838,-176.789,6.701,148.290
C05124=1217.103,268.321,-63.866,-176.787,6.703,148.289
C05125=1217.098,268.571,-63.894,-176.784,6.705,148.289
C05126=1217.094,268.819,-63.922,-176.782,6.707,148.289
C05127=1217.089,269.067,-63.949,-176.779,6.710,148.289
C05128=1217.086,269.316,-63.977,-176.777,6.712,148.289
C05129=1217.081,269.564,-64.005,-176.774,6.714,148.288
C05130=1217.077,269.812,-64.032,-176.772,6.716,148.288
C05131=1217.073,270.061,-64.060,-176.769,6.719,148.288
C05132=1217.068,270.310,-64.088,-176.767,6.721,148.288
C05133=1217.063,270.558,-64.115,-176.765,6.723,148.288
C05134=1217.059,270.807,-64.143,-176.762,6.725,148.288
C05135=1217.055,271.055,-64.171,-176.759,6.728,148.288
C05136=1217.050,271.302,-64.198,-176.757,6.730,148.287
C05137=1217.046,271.552,-64.226,-176.755,6.732,148.287
C05138=1217.041,271.800,-64.254,-176.751,6.735,148.287
C05139=1217.038,272.048,-64.282,-176.749,6.737,148.287
C05140=1217.033,272.297,-64.309,-176.747,6.739,148.287
C05141=1217.028,272.545,-64.337,-176.745,6.741,148.287
C05142=1217.024,272.794,-64.366,-176.741,6.744,148.286
C05143=1217.020,273.042,-64.394,-176.739,6.746,148.286
C05144=1217.015,273.290,-64.421,-176.737,6.748,148.286
C05145=1217.011,273.539,-64.449,-176.735,6.750,148.286
C05146=1217.006,273.787,-64.477,-176.732,6.753,148.286
C05147=1217.002,274.035,-64.505,-176.729,6.755,148.286
C05148=1216.998,274.284,-64.532,-176.727,6.757,148.285
C05149=1216.993,274.533,-64.561,-176.724,6.760,148.285
C05150=1216.989,274.781,-64.589,-176.722,6.762,148.285
C05151=1216.985,275.029,-64.617,-176.720,6.764,148.285
C05152=1216.980,275.277,-64.646,-176.717,6.767,148.285
C05153=1216.975,275.526,-64.673,-176.714,6.769,148.285
C05154=1216.972,275.774,-64.701,-176.712,6.771,148.284
C05155=1216.967,276.023,-64.729,-176.710,6.773,148.284
C05156=1216.963,276.271,-64.757,-176.707,6.776,148.284
C05157=1216.958,276.519,-64.785,-176.704,6.778,148.284
C05158=1216.954,276.768,-64.814,-176.702,6.781,148.284
C05159=1216.950,277.016,-64.842,-176.699,6.783,148.284
C05160=1216.946,277.264,-64.870,-176.697,6.785,148.284
C05161=1216.941,277.513,-64.897,-176.694,6.787,148.283
C05162=1216.937,277.762,-64.925,-176.692,6.790,148.283
C05163=1216.932,278.010,-64.954,-176.690,6.793,148.283
C05164=1216.927,278.258,-64.982,-176.687,6.794,148.283
C05165=1216.924,278.506,-65.010,-176.685,6.797,148.283
C05166=1216.918,278.755,-65.038,-176.682,6.799,148.283
C05167=1216.915,279.003,-65.066,-176.680,6.802,148.283
C05168=1216.910,279.252,-65.095,-176.677,6.804,148.283
C05169=1216.906,279.500,-65.123,-176.674,6.807,148.282
C05170=1216.901,279.749,-65.152,-176.672,6.809,148.282
C05171=1216.897,279.997,-65.179,-176.670,6.811,148.282
C05172=1216.893,280.245,-65.207,-176.667,6.814,148.282
C05173=1216.889,280.493,-65.237,-176.665,6.816,148.282
C05174=1216.885,280.741,-65.265,-176.663,6.818,148.282
C05175=1216.880,280.990,-65.293,-176.659,6.821,148.281
C05176=1216.876,281.238,-65.321,-176.657,6.823,148.281
C05177=1216.871,281.486,-65.350,-176.655,6.825,148.281
C05178=1216.867,281.735,-65.378,-176.652,6.828,148.281
C05179=1216.862,281.983,-65.406,-176.650,6.830,148.281
C05180=1216.858,282.232,-65.434,-176.647,6.832,148.281
C05181=1216.854,282.480,-65.464,-176.645,6.835,148.281
C05182=1216.849,282.728,-65.492,-176.643,6.837,148.281
C05183=1216.845,282.977,-65.520,-176.640,6.839,148.280
C05184=1216.840,283.225,-65.549,-176.637,6.842,148.280
C05185=1216.836,283.474,-65.577,-176.635,6.844,148.280
C05186=1216.832,283.722,-65.606,-176.633,6.846,148.280
C05187=1216.828,283.970,-65.634,-176.630,6.849,148.280
C05188=1216.823,284.219,-65.663,-176.628,6.851,148.280
C05189=1216.818,284.467,-65.691,-176.626,6.854,148.280
C05190=1216.815,284.715,-65.720,-176.622,6.856,148.280
C05191=1216.810,284.964,-65.749,-176.620,6.859,148.280
C05192=1216.805,285.212,-65.777,-176.618,6.862,148.279
C05193=1216.802,285.460,-65.805,-176.615,6.863,148.279
C05194=1216.797,285.708,-65.834,-176.613,6.866,148.279
C05195=1216.793,285.957,-65.862,-176.610,6.869,148.279
C05196=1216.788,286.205,-65.891,-176.608,6.871,148.279
C05197=1216.784,286.453,-65.920,-176.606,6.873,148.279
C05198=1216.780,286.702,-65.948,-176.603,6.876,148.279
C05199=1216.775,286.950,-65.977,-176.601,6.878,148.279
C05200=1216.771,287.198,-66.006,-176.598,6.880,148.278
C05201=1216.767,287.447,-66.034,-176.595,6.883,148.278
C05202=1216.763,287.695,-66.064,-176.593,6.885,148.278
C05203=1216.758,287.943,-66.092,-176.591,6.887,148.278
C05204=1216.753,288.191,-66.122,-176.588,6.890,148.278
C05205=1216.750,288.440,-66.150,-176.586,6.892,148.278
C05206=1216.745,288.688,-66.178,-176.583,6.895,148.278
C05207=1216.740,288.962,-66.210,-176.581,6.897,148.278
C05208=1216.735,289.236,-66.242,-176.578,6.900,148.278
C05209=1216.731,289.511,-66.274,-176.575,6.903,148.278
C05210=1216.726,289.785,-66.305,-176.572,6.906,148.277
C05211=1216.722,290.033,-66.335,-176.570,6.908,148.277
C05212=1216.717,290.281,-66.364,-176.568,6.910,148.277
C05213=1216.712,290.530,-66.393,-176.565,6.913,148.277
C05214=1216.709,290.778,-66.422,-176.563,6.915,148.277
C05215=1216.704,291.026,-66.450,-176.561,6.918,148.277
C05216=1216.700,291.274,-66.479,-176.558,6.921,148.277
C05217=1216.695,291.523,-66.508,-176.556,6.923,148.277
C05218=1216.691,291.771,-66.538,-176.553,6.926,148.277
C05219=1216.687,292.019,-66.566,-176.550,6.928,148.276
C05220=1216.682,292.267,-66.595,-176.548,6.930,148.276
C05221=1216.678,292.516,-66.624,-176.546,6.933,148.276
C05222=1216.674,292.764,-66.654,-176.544,6.935,148.276
C05223=1216.670,293.013,-66.682,-176.540,6.938,148.276
C05224=1216.665,293.261,-66.712,-176.538,6.940,148.276
C05225=1216.661,293.509,-66.741,-176.536,6.942,148.276
C05226=1216.656,293.757,-66.770,-176.533,6.945,148.276
C05227=1216.653,294.005,-66.799,-176.531,6.948,148.276
C05228=1216.648,294.254,-66.828,-176.528,6.950,148.276
C05229=1216.643,294.502,-66.856,-176.526,6.953,148.276
C05230=1216.639,294.750,-66.886,-176.524,6.955,148.276
C05231=1216.635,294.998,-66.915,-176.521,6.958,148.276
C05232=1216.631,295.247,-66.945,-176.519,6.960,148.275
C05233=1216.626,295.496,-66.973,-176.516,6.963,148.275
C05234=1216.622,295.744,-67.003,-176.514,6.965,148.275
C05235=1216.617,295.991,-67.032,-176.512,6.967,148.275
C05236=1216.613,296.240,-67.061,-176.509,6.970,148.275
C05237=1216.609,296.488,-67.091,-176.507,6.972,148.275
C05238=1216.605,296.736,-67.120,-176.504,6.975,148.275
C05239=1216.600,296.985,-67.149,-176.502,6.978,148.275
C05240=1216.596,297.233,-67.179,-176.500,6.980,148.275
C05241=1216.591,297.481,-67.208,-176.497,6.983,148.275
C05242=1216.587,297.729,-67.237,-176.495,6.985,148.275
C05243=1216.583,297.977,-67.267,-176.492,6.988,148.275
C05244=1216.579,298.226,-67.296,-176.490,6.990,148.275
C05245=1216.575,298.474,-67.325,-176.487,6.993,148.274
C05246=1216.570,298.722,-67.355,-176.485,6.995,148.274
C05247=1216.566,298.971,-67.384,-176.483,6.997,148.274
C05248=1216.561,299.218,-67.413,-176.480,7.000,148.274
C05249=1216.557,299.466,-67.443,-176.478,7.003,148.274
C05250=1216.553,299.715,-67.472,-176.475,7.005,148.274
C05251=1216.549,299.963,-67.502,-176.473,7.008,148.274
C05252=1216.545,300.211,-67.531,-176.470,7.011,148.274
C05253=1216.541,300.459,-67.561,-176.468,7.013,148.274
C05254=1216.536,300.708,-67.590,-176.466,7.015,148.274
C05255=1216.531,300.956,-67.620,-176.463,7.018,148.274
C05256=1216.527,301.205,-67.650,-176.461,7.020,148.274
C05257=1216.523,301.453,-67.679,-176.459,7.023,148.274
C05258=1216.519,301.701,-67.709,-176.457,7.026,148.274
C05259=1216.514,301.949,-67.738,-176.454,7.029,148.274
C05260=1216.510,302.197,-67.767,-176.452,7.031,148.274
C05261=1216.506,302.445,-67.797,-176.450,7.033,148.274
C05262=1216.501,302.694,-67.827,-176.447,7.036,148.274
C05263=1216.497,302.942,-67.856,-176.445,7.038,148.274
C05264=1216.493,303.190,-67.886,-176.442,7.041,148.274
C05265=1216.489,303.438,-67.916,-176.440,7.043,148.273
C05266=1216.484,303.686,-67.945,-176.437,7.046,148.273
C05267=1216.480,303.934,-67.975,-176.435,7.048,148.273
C05268=1216.475,304.183,-68.005,-176.432,7.051,148.273
C05269=1216.471,304.431,-68.034,-176.430,7.054,148.273
C05270=1216.467,304.679,-68.064,-176.428,7.056,148.273
C05271=1216.463,304.927,-68.094,-176.425,7.059,148.273
C05272=1216.458,305.176,-68.124,-176.423,7.061,148.273
C05273=1216.454,305.424,-68.153,-176.420,7.064,148.273
C05274=1216.450,305.672,-68.183,-176.418,7.066,148.273
C05275=1216.446,305.920,-68.213,-176.416,7.069,148.273
C05276=1216.441,306.169,-68.243,-176.414,7.072,148.273
C05277=1216.437,306.417,-68.272,-176.411,7.075,148.273
C05278=1216.433,306.664,-68.303,-176.409,7.077,148.273
C05279=1216.428,306.913,-68.333,-176.407,7.079,148.273
C05280=1216.424,307.161,-68.362,-176.404,7.082,148.273
C05281=1216.420,307.409,-68.392,-176.402,7.084,148.273
C05282=1216.415,307.658,-68.422,-176.400,7.088,148.273
C05283=1216.411,307.905,-68.452,-176.398,7.090,148.273
C05284=1216.407,308.153,-68.482,-176.395,7.093,148.273
C05285=1216.402,308.402,-68.512,-176.393,7.095,148.273
C05286=1216.398,308.650,-68.542,-176.390,7.098,148.273
C05287=1216.394,308.898,-68.572,-176.388,7.100,148.273
C05288=1216.389,309.146,-68.602,-176.385,7.103,148.273
C05289=1216.385,309.394,-68.632,-176.383,7.106,148.273
C05290=1216.382,309.643,-68.662,-176.380,7.109,148.273
C05291=1216.377,309.891,-68.692,-176.378,7.111,148.273
C05292=1216.373,310.139,-68.722,-176.376,7.113,148.273
C05293=1216.368,310.387,-68.753,-176.374,7.116,148.273
C05294=1216.364,310.636,-68.782,-176.371,7.118,148.272
C05295=1216.360,310.883,-68.812,-176.369,7.121,148.272
C05296=1216.355,311.132,-68.842,-176.367,7.124,148.273
C05297=1216.351,311.379,-68.872,-176.364,7.127,148.273
C05298=1216.347,311.627,-68.903,-176.362,7.129,148.273
C05299=1216.343,311.876,-68.933,-176.360,7.132,148.273
C05300=1216.338,312.124,-68.963,-176.358,7.134,148.273
C05301=1216.334,312.373,-68.993,-176.355,7.137,148.273
C05302=1216.330,312.621,-69.024,-176.353,7.140,148.272
C05303=1216.326,312.869,-69.053,-176.350,7.143,148.272
C05304=1216.321,313.117,-69.084,-176.348,7.145,148.273
C05305=1216.317,313.364,-69.114,-176.346,7.148,148.273
C05306=1216.313,313.613,-69.144,-176.344,7.151,148.273
C05307=1216.308,313.861,-69.175,-176.341,7.154,148.273
C05308=1216.304,314.109,-69.206,-176.339,7.156,148.273
C05309=1216.300,314.358,-69.235,-176.337,7.158,148.272
C05310=1216.296,314.606,-69.266,-176.334,7.161,148.272
C05311=1216.292,314.881,-69.300,-176.332,7.164,148.273
C05312=1216.286,315.157,-69.333,-176.329,7.167,148.273
C05313=1216.282,315.433,-69.367,-176.327,7.170,148.273
C05314=1216.277,315.709,-69.400,-176.324,7.173,148.273
C05315=1216.273,315.957,-69.431,-176.322,7.176,148.273
C05316=1216.268,316.205,-69.462,-176.320,7.178,148.273
C05317=1216.264,316.453,-69.492,-176.317,7.181,148.273
C05318=1216.260,316.702,-69.523,-176.315,7.184,148.273
C05319=1216.256,316.950,-69.553,-176.313,7.187,148.273
C05320=1216.251,317.198,-69.583,-176.311,7.189,148.273
C05321=1216.247,317.446,-69.614,-176.308,7.192,148.273
C05322=1216.243,317.693,-69.644,-176.306,7.194,148.273
C05323=1216.239,317.943,-69.675,-176.304,7.197,148.273
C05324=1216.235,318.190,-69.705,-176.302,7.200,148.273
C05325=1216.230,318.438,-69.736,-176.299,7.203,148.273
C05326=1216.225,318.686,-69.766,-176.297,7.205,148.273
C05327=1216.222,318.935,-69.797,-176.295,7.208,148.273
C05328=1216.218,319.183,-69.828,-176.292,7.210,148.273
C05329=1216.213,319.431,-69.859,-176.290,7.213,148.273
C05330=1216.209,319.678,-69.889,-176.288,7.216,148.273
C05331=1216.205,319.927,-69.920,-176.285,7.219,148.273
C05332=1216.200,320.175,-69.951,-176.283,7.221,148.273
C05333=1216.196,320.423,-69.981,-176.281,7.224,148.273
C05334=1216.192,320.670,-70.012,-176.279,7.227,148.273
C05335=1216.188,320.919,-70.043,-176.276,7.230,148.273
C05336=1216.183,321.167,-70.073,-176.274,7.232,148.273
C05337=1216.179,321.415,-70.104,-176.273,7.235,148.273
C05338=1216.175,321.663,-70.135,-176.270,7.238,148.273
C05339=1216.171,321.911,-70.166,-176.268,7.240,148.273
C05340=1216.166,322.159,-70.196,-176.266,7.243,148.274
C05341=1216.163,322.408,-70.227,-176.264,7.245,148.273
C05342=1216.158,322.656,-70.258,-176.261,7.248,148.273
C05343=1216.154,322.903,-70.288,-176.259,7.251,148.274
C05344=1216.150,323.152,-70.319,-176.257,7.254,148.274
C05345=1216.145,323.400,-70.350,-176.254,7.256,148.274
C05346=1216.141,323.648,-70.380,-176.252,7.260,148.274
C05347=1216.137,323.896,-70.412,-176.250,7.262,148.274
C05348=1216.133,324.144,-70.443,-176.247,7.265,148.274
C05349=1216.128,324.392,-70.474,-176.246,7.267,148.274
C05350=1216.124,324.640,-70.505,-176.243,7.270,148.274
C05351=1216.120,324.888,-70.535,-176.241,7.273,148.274
C05352=1216.116,325.136,-70.566,-176.239,7.276,148.274
C05353=1216.112,325.385,-70.597,-176.237,7.278,148.274
C05354=1216.107,325.632,-70.628,-176.235,7.282,148.274
C05355=1216.103,325.880,-70.659,-176.232,7.284,148.274
C05356=1216.099,326.129,-70.690,-176.230,7.287,148.274
C05357=1216.094,326.377,-70.721,-176.228,7.289,148.274
C05358=1216.091,326.624,-70.752,-176.225,7.292,148.274
C05359=1216.087,326.872,-70.783,-176.224,7.295,148.275
C05360=1216.082,327.120,-70.814,-176.221,7.298,148.275
C05361=1216.078,327.369,-70.845,-176.219,7.300,148.275
C05362=1216.074,327.616,-70.876,-176.217,7.303,148.275
C05363=1216.070,327.865,-70.908,-176.215,7.306,148.275
C05364=1216.065,328.113,-70.938,-176.213,7.309,148.275
C05365=1216.061,328.360,-70.970,-176.210,7.311,148.275
C05366=1216.057,328.609,-71.001,-176.208,7.315,148.275
C05367=1216.052,328.857,-71.032,-176.206,7.317,148.275
C05368=1216.048,329.105,-71.064,-176.204,7.320,148.275
C05369=1216.044,329.353,-71.094,-176.202,7.322,148.275
C05370=1216.040,329.600,-71.126,-176.200,7.326,148.276
C05371=1216.036,329.849,-71.157,-176.197,7.328,148.275
C05372=1216.031,330.097,-71.188,-176.195,7.331,148.276
C05373=1216.027,330.345,-71.220,-176.193,7.334,148.276
C05374=1216.023,330.593,-71.250,-176.191,7.337,148.276
C05375=1216.019,330.841,-71.282,-176.189,7.339,148.276
C05376=1216.014,331.089,-71.313,-176.187,7.342,148.276
C05377=1216.011,331.337,-71.345,-176.185,7.345,148.276
C05378=1216.006,331.585,-71.376,-176.183,7.347,148.276
C05379=1216.002,331.833,-71.407,-176.181,7.351,148.276
C05380=1215.998,332.081,-71.438,-176.179,7.353,148.276
C05381=1215.994,332.329,-71.470,-176.176,7.356,148.277
C05382=1215.989,332.577,-71.501,-176.174,7.358,148.277
C05383=1215.986,332.825,-71.533,-176.172,7.362,148.277
C05384=1215.981,333.073,-71.563,-176.170,7.364,148.277
C05385=1215.977,333.321,-71.595,-176.168,7.367,148.277
C05386=1215.972,333.568,-71.627,-176.166,7.370,148.277
C05387=1215.968,333.817,-71.658,-176.163,7.373,148.277
C05388=1215.964,334.064,-71.690,-176.162,7.375,148.277
C05389=1215.960,334.313,-71.721,-176.160,7.379,148.278
C05390=1215.956,334.560,-71.753,-176.158,7.381,148.277
C05391=1215.952,334.808,-71.784,-176.155,7.384,148.278
C05392=1215.947,335.056,-71.815,-176.153,7.386,148.278
C05393=1215.944,335.304,-71.847,-176.151,7.390,148.278
C05394=1215.939,335.552,-71.879,-176.149,7.392,148.278
C05395=1215.935,335.801,-71.910,-176.147,7.395,148.278
C05396=1215.930,336.048,-71.942,-176.145,7.398,148.278
C05397=1215.927,336.296,-71.974,-176.143,7.401,148.278
C05398=1215.922,336.544,-72.004,-176.141,7.403,148.278
C05399=1215.917,336.792,-72.037,-176.139,7.407,148.279
C05400=1215.914,337.040,-72.069,-176.137,7.409,148.279
C05401=1215.909,337.288,-72.100,-176.135,7.412,148.279
C05402=1215.905,337.536,-72.131,-176.133,7.415,148.279
C05403=1215.901,337.784,-72.163,-176.131,7.417,148.279
C05404=1215.897,338.032,-72.195,-176.129,7.421,148.279
C05405=1215.892,338.279,-72.227,-176.127,7.423,148.279
C05406=1215.889,338.527,-72.258,-176.124,7.426,148.280
C05407=1215.885,338.776,-72.290,-176.123,7.429,148.280
C05408=1215.880,339.024,-72.322,-176.120,7.432,148.280
C05409=1215.876,339.272,-72.353,-176.119,7.434,148.280
C05410=1215.872,339.520,-72.385,-176.116,7.438,148.280
C05411=1215.868,339.767,-72.417,-176.115,7.440,148.280
C05412=1215.863,340.016,-72.449,-176.112,7.443,148.280
C05413=1215.859,340.263,-72.481,-176.110,7.446,148.281
C05414=1215.855,340.512,-72.512,-176.108,7.449,148.281
C05415=1215.850,340.789,-72.548,-176.107,7.452,148.281
C05416=1215.846,341.067,-72.584,-176.104,7.455,148.281
C05417=1215.841,341.345,-72.620,-176.102,7.458,148.281
C05418=1215.836,341.623,-72.655,-176.099,7.462,148.281
C05419=1215.832,341.871,-72.687,-176.097,7.465,148.282
C05420=1215.828,342.119,-72.719,-176.096,7.467,148.282
C05421=1215.824,342.367,-72.751,-176.093,7.471,148.282
C05422=1215.819,342.615,-72.783,-176.091,7.473,148.282
C05423=1215.815,342.863,-72.815,-176.090,7.475,148.282
C05424=1215.811,343.110,-72.846,-176.087,7.479,148.282
C05425=1215.807,343.359,-72.879,-176.086,7.481,148.283
C05426=1215.803,343.607,-72.911,-176.084,7.485,148.283
C05427=1215.798,343.854,-72.943,-176.082,7.487,148.283
C05428=1215.794,344.102,-72.974,-176.080,7.491,148.283
C05429=1215.791,344.351,-73.006,-176.078,7.493,148.283
C05430=1215.786,344.598,-73.039,-176.076,7.496,148.284
C05431=1215.782,344.846,-73.071,-176.074,7.499,148.284
C05432=1215.778,345.094,-73.103,-176.072,7.501,148.284
C05433=1215.774,345.342,-73.135,-176.070,7.505,148.284
C05434=1215.769,345.590,-73.167,-176.068,7.507,148.284
C05435=1215.765,345.838,-73.199,-176.066,7.510,148.284
C05436=1215.761,346.086,-73.232,-176.065,7.513,148.285
C05437=1215.756,346.333,-73.263,-176.062,7.516,148.285
C05438=1215.752,346.581,-73.296,-176.061,7.519,148.285
C05439=1215.749,346.829,-73.328,-176.059,7.522,148.285
C05440=1215.744,347.077,-73.361,-176.057,7.525,148.285
C05441=1215.740,347.325,-73.392,-176.055,7.527,148.286
C05442=1215.735,347.573,-73.424,-176.053,7.531,148.286
C05443=1215.732,347.821,-73.457,-176.051,7.533,148.286
C05444=1215.728,348.069,-73.489,-176.049,7.536,148.286
C05445=1215.723,348.316,-73.521,-176.048,7.539,148.286
C05446=1215.719,348.565,-73.553,-176.045,7.542,148.287
C05447=1215.715,348.812,-73.586,-176.044,7.545,148.287
C05448=1215.711,349.060,-73.618,-176.042,7.547,148.287
C05449=1215.707,349.308,-73.650,-176.040,7.551,148.287
C05450=1215.703,349.555,-73.683,-176.038,7.553,148.287
C05451=1215.698,349.804,-73.715,-176.036,7.557,148.288
C05452=1215.694,350.052,-73.747,-176.034,7.559,148.288
C05453=1215.690,350.299,-73.780,-176.032,7.562,148.288
C05454=1215.686,350.547,-73.812,-176.031,7.565,148.288
C05455=1215.681,350.795,-73.844,-176.029,7.568,148.289
C05456=1215.677,351.043,-73.878,-176.027,7.571,148.289
C05457=1215.674,351.291,-73.909,-176.025,7.574,148.289
C05458=1215.669,351.539,-73.941,-176.023,7.577,148.289
C05459=1215.665,351.786,-73.974,-176.022,7.579,148.289
C05460=1215.661,352.034,-74.006,-176.019,7.583,148.290
C05461=1215.657,352.282,-74.040,-176.018,7.585,148.290
C05462=1215.653,352.530,-74.071,-176.016,7.588,148.290
C05463=1215.649,352.778,-74.105,-176.014,7.592,148.290
C05464=1215.644,353.026,-74.137,-176.013,7.594,148.291
C05465=1215.640,353.274,-74.169,-176.011,7.597,148.291
C05466=1215.636,353.521,-74.202,-176.009,7.600,148.291
C05467=1215.631,353.770,-74.234,-176.007,7.602,148.291
C05468=1215.628,354.017,-74.267,-176.005,7.606,148.291
C05469=1215.624,354.265,-74.299,-176.004,7.609,148.292
C05470=1215.619,354.513,-74.332,-176.002,7.612,148.292
C05471=1215.615,354.761,-74.364,-176.000,7.614,148.292
